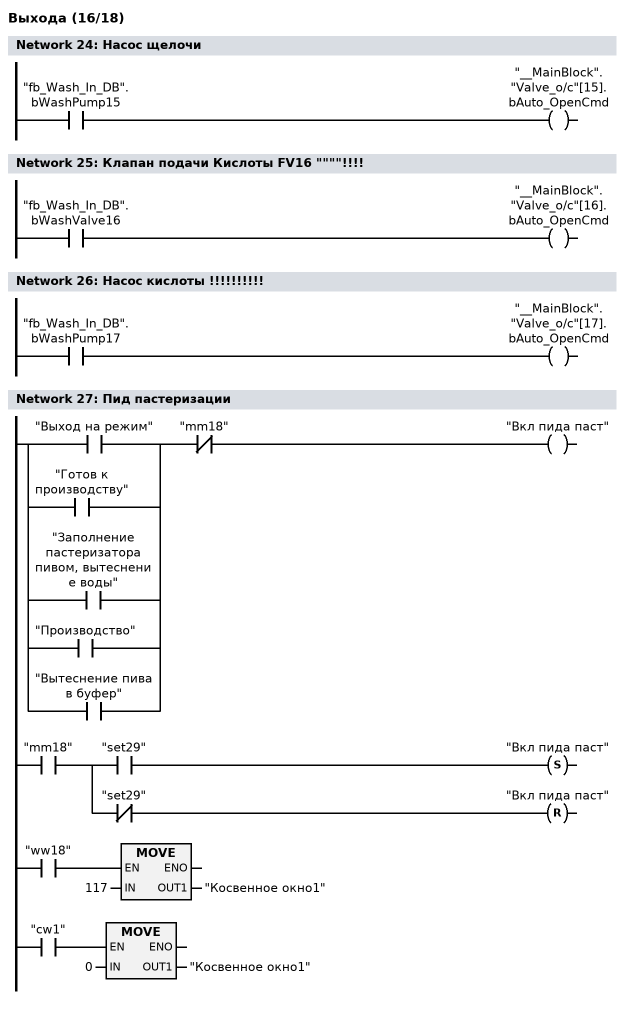
   RUNG wire#powerrail
      Contact( "fb_Wash_In_DB".bWashPump15 )
      Coil( "__MainBlock"."Valve_o/c"[15].bAuto_OpenCmd )
   END_RUNG
   // the same network as SCL:
   "__MainBlock"."Valve_o/c"[15].bAuto_OpenCmd := "fb_Wash_In_DB".bWashPump15;
END_REGION

REGION Network 25: Клапан подачи Кислоты FV16 """"!!!!
   RUNG wire#powerrail
      Contact( "fb_Wash_In_DB".bWashValve16 )
      Coil( "__MainBlock"."Valve_o/c"[16].bAuto_OpenCmd )
   END_RUNG
   // the same network as SCL:
   "__MainBlock"."Valve_o/c"[16].bAuto_OpenCmd := "fb_Wash_In_DB".bWashValve16;
END_REGION

REGION Network 26: Насос кислоты !!!!!!!!!!
   RUNG wire#powerrail
      Contact( "fb_Wash_In_DB".bWashPump17 )
      Coil( "__MainBlock"."Valve_o/c"[17].bAuto_OpenCmd )
   END_RUNG
   // the same network as SCL:
   "__MainBlock"."Valve_o/c"[17].bAuto_OpenCmd := "fb_Wash_In_DB".bWashPump17;
END_REGION

REGION Network 27: Пид пастеризации
   RUNG wire#powerrail
      Contact( "Выход на режим" )
      wire#w1
      I_Contact( "mm18" )
      Coil( "Вкл пида паст" )
   END_RUNG
   RUNG wire#powerrail
      Contact( "Готов к производству" )
   END_RUNG wire#w1
   RUNG wire#powerrail
      Contact( "Заполнение пастеризатора пивом, вытеснение воды" )
   END_RUNG wire#w1
   RUNG wire#powerrail
      Contact( "Производство" )
   END_RUNG wire#w1
   RUNG wire#powerrail
      Contact( "Вытеснение пива в буфер" )
   END_RUNG wire#w1
   RUNG wire#powerrail
      Contact( "mm18" )
      wire#w2
      Contact( "set29" )
      S_Coil( "Вкл пида паст" )
   END_RUNG
   RUNG wire#w2
      I_Contact( "set29" )
      R_Coil( "Вкл пида паст" )
   END_RUNG
   RUNG wire#powerrail
      Contact( "ww18" )
      Move(in := 117, out1 => "Косвенное окно1")
   END_RUNG
   RUNG wire#powerrail
      Contact( "cw1" )
      Move(in := 0, out1 => "Косвенное окно1")
   END_RUNG
   // the same network as SCL:
   "Вкл пида паст" := ("Выход на режим" OR "Готов к производству" OR "Заполнение пастеризатора пивом, вытеснение воды" OR "Производство" OR "Вытеснение пива в буфер") AND NOT "mm18";
   IF "mm18" AND "set29" THEN "Вкл пида паст" := TRUE; END_IF;
   IF "mm18" AND NOT "set29" THEN "Вкл пида паст" := FALSE; END_IF;
   IF "ww18" THEN "Косвенное окно1" := 117; END_IF;
   IF "cw1" THEN "Косвенное окно1" := 0; END_IF;
END_REGION

REGION Network 28: Пид охлаждения
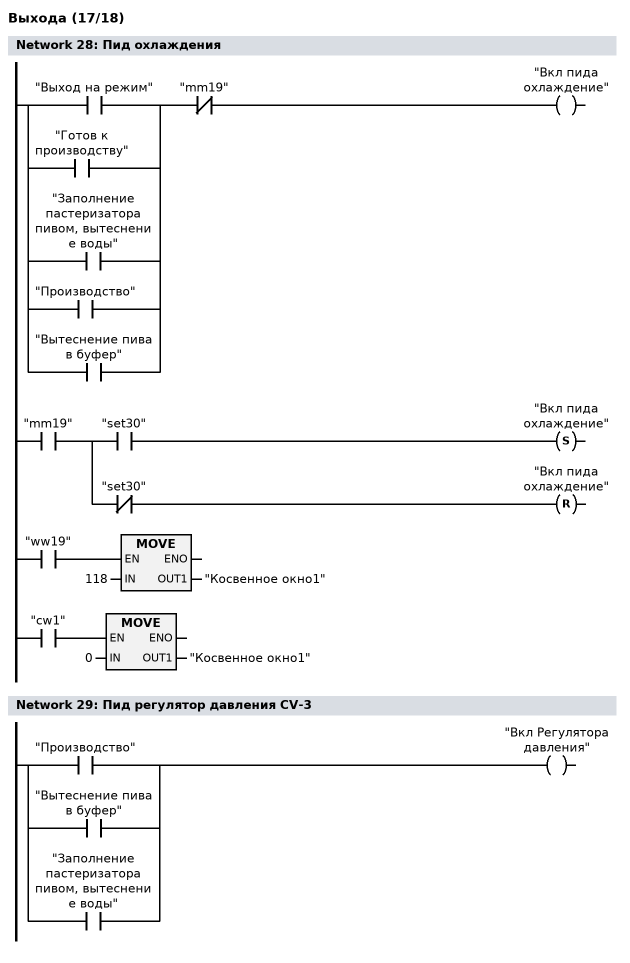
   RUNG wire#powerrail
      Contact( "Выход на режим" )
      wire#w1
      I_Contact( "mm19" )
      Coil( "Вкл пида охлаждение" )
   END_RUNG
   RUNG wire#powerrail
      Contact( "Готов к производству" )
   END_RUNG wire#w1
   RUNG wire#powerrail
      Contact( "Заполнение пастеризатора пивом, вытеснение воды" )
   END_RUNG wire#w1
   RUNG wire#powerrail
      Contact( "Производство" )
   END_RUNG wire#w1
   RUNG wire#powerrail
      Contact( "Вытеснение пива в буфер" )
   END_RUNG wire#w1
   RUNG wire#powerrail
      Contact( "mm19" )
      wire#w2
      Contact( "set30" )
      S_Coil( "Вкл пида охлаждение" )
   END_RUNG
   RUNG wire#w2
      I_Contact( "set30" )
      R_Coil( "Вкл пида охлаждение" )
   END_RUNG
   RUNG wire#powerrail
      Contact( "ww19" )
      Move(in := 118, out1 => "Косвенное окно1")
   END_RUNG
   RUNG wire#powerrail
      Contact( "cw1" )
      Move(in := 0, out1 => "Косвенное окно1")
   END_RUNG
   // the same network as SCL:
   "Вкл пида охлаждение" := ("Выход на режим" OR "Готов к производству" OR "Заполнение пастеризатора пивом, вытеснение воды" OR "Производство" OR "Вытеснение пива в буфер") AND NOT "mm19";
   IF "mm19" AND "set30" THEN "Вкл пида охлаждение" := TRUE; END_IF;
   IF "mm19" AND NOT "set30" THEN "Вкл пида охлаждение" := FALSE; END_IF;
   IF "ww19" THEN "Косвенное окно1" := 118; END_IF;
   IF "cw1" THEN "Косвенное окно1" := 0; END_IF;
END_REGION

REGION Network 29: Пид регулятор давления CV-3
   RUNG wire#powerrail
      Contact( "Производство" )
      wire#w1
      Coil( "Вкл Регулятора давления" )
   END_RUNG
   RUNG wire#powerrail
      Contact( "Вытеснение пива в буфер" )
   END_RUNG wire#w1
   RUNG wire#powerrail
      Contact( "Заполнение пастеризатора пивом, вытеснение воды" )
   END_RUNG wire#w1
   // the same network as SCL:
   "Вкл Регулятора давления" := "Производство" OR "Вытеснение пива в буфер" OR "Заполнение пастеризатора пивом, вытеснение воды";
END_REGION

REGION Network 30: Пид произовдительности М1=М2
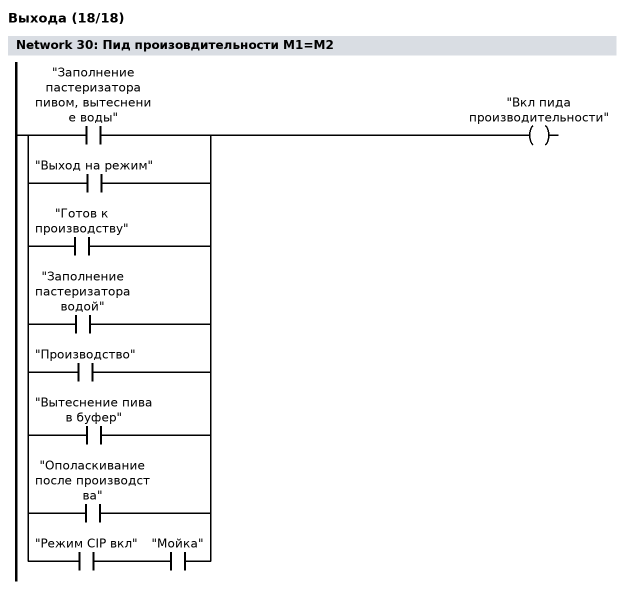
   RUNG wire#powerrail
      Contact( "Заполнение пастеризатора пивом, вытеснение воды" )
      wire#w1
      Coil( "Вкл пида производительности" )
   END_RUNG
   RUNG wire#powerrail
      Contact( "Выход на режим" )
   END_RUNG wire#w1
   RUNG wire#powerrail
      Contact( "Готов к производству" )
   END_RUNG wire#w1
   RUNG wire#powerrail
      Contact( "Заполнение пастеризатора водой" )
   END_RUNG wire#w1
   RUNG wire#powerrail
      Contact( "Производство" )
   END_RUNG wire#w1
   RUNG wire#powerrail
      Contact( "Вытеснение пива в буфер" )
   END_RUNG wire#w1
   RUNG wire#powerrail
      Contact( "Ополаскивание после производства" )
   END_RUNG wire#w1
   RUNG wire#powerrail
      Contact( "Режим СIP вкл" )
      Contact( "Мойка" )
   END_RUNG wire#w1
   // the same network as SCL:
   "Вкл пида производительности" := "Заполнение пастеризатора пивом, вытеснение воды" OR "Выход на режим" OR "Готов к производству" OR "Заполнение пастеризатора водой" OR "Производство" OR "Вытеснение пива в буфер" OR "Ополаскивание после производства" OR ("Режим СIP вкл" AND "Мойка");
END_REGION
END_ORGANIZATION_BLOCK

ORGANIZATION_BLOCK "Реж_Пастеризация пива"   // OB126, LAD, ProgramCycle
TITLE = "Main Program Sweep (Cycle)"
{ S7_Optimized_Access := 'TRUE' }
VERSION : 0.1
   VAR_INPUT
      Initial_Call : Bool;   // Initial call of this OB
      Remanence : Bool;   // =True, if remanent data are available
   END_VAR
BEGIN

REGION Network 1: Заполнение пивом
   // временно привязал переменные на прямую без обработки сигналов DI - ИСПРАВИТЬ!!!!!
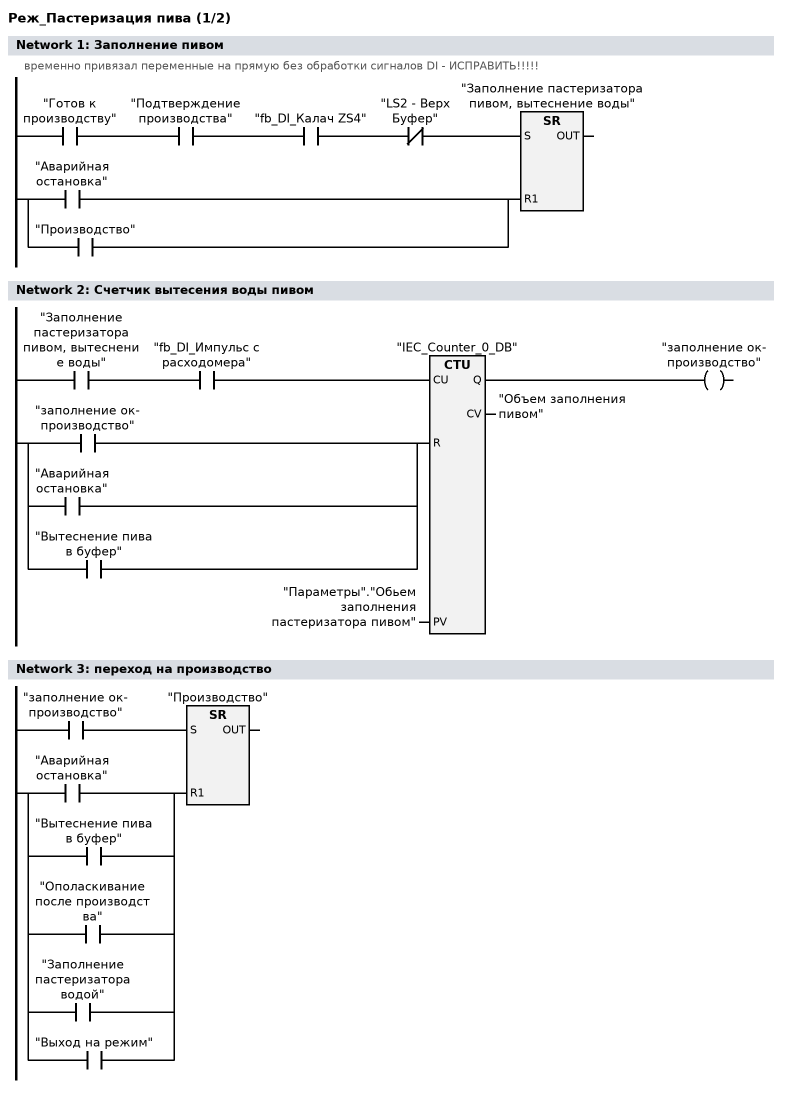
   RUNG wire#powerrail
      Contact( "Готов к производству" )
      Contact( "Подтверждение производства" )
      Contact( "fb_DI_Калач ZS4" )
      I_Contact( "LS2 - Верх Буфер" )
      S_SR(operand := "Заполнение пастеризатора пивом, вытеснение воды", r1 := wire#w1)
   END_RUNG
   RUNG wire#powerrail
      Contact( "Аварийная остановка" )
   END_RUNG wire#w1
   RUNG wire#powerrail
      Contact( "Производство" )
   END_RUNG wire#w1
   // the same network as SCL:
   IF "Готов к производству" AND "Подтверждение производства" AND "fb_DI_Калач ZS4" AND NOT "LS2 - Верх Буфер" THEN
       "Заполнение пастеризатора пивом, вытеснение воды" := TRUE;   // SR flip-flop
   END_IF;
   IF "Аварийная остановка" OR "Производство" THEN
       "Заполнение пастеризатора пивом, вытеснение воды" := FALSE;
   END_IF;
END_REGION

REGION Network 2: Счетчик вытесения воды пивом
   "IEC_Counter_0_DB".CTU(CU := "Заполнение пастеризатора пивом, вытеснение воды" AND "fb_DI_Импульс с расходомера",
                          R := "заполнение ок- производство" OR "Аварийная остановка" OR "Вытеснение пива в буфер",
                          PV := "Параметры"."Обьем заполнения пастеризатора пивом",
                          CV => "Объем заполнения пивом");
   "заполнение ок- производство" := "IEC_Counter_0_DB".Q;
END_REGION

REGION Network 3: переход на производство
   RUNG wire#powerrail
      Contact( "заполнение ок- производство" )
      S_SR(operand := "Производство", r1 := wire#w1)
   END_RUNG
   RUNG wire#powerrail
      Contact( "Аварийная остановка" )
   END_RUNG wire#w1
   RUNG wire#powerrail
      Contact( "Вытеснение пива в буфер" )
   END_RUNG wire#w1
   RUNG wire#powerrail
      Contact( "Ополаскивание после производства" )
   END_RUNG wire#w1
   RUNG wire#powerrail
      Contact( "Заполнение пастеризатора водой" )
   END_RUNG wire#w1
   RUNG wire#powerrail
      Contact( "Выход на режим" )
   END_RUNG wire#w1
   // the same network as SCL:
   IF "заполнение ок- производство" THEN
       "Производство" := TRUE;   // SR flip-flop
   END_IF;
   IF "Аварийная остановка" OR "Вытеснение пива в буфер" OR "Ополаскивание после производства" OR "Заполнение пастеризатора водой" OR "Выход на режим" THEN
       "Производство" := FALSE;
   END_IF;
END_REGION

REGION Network 4: Счетчик объема пастеризации
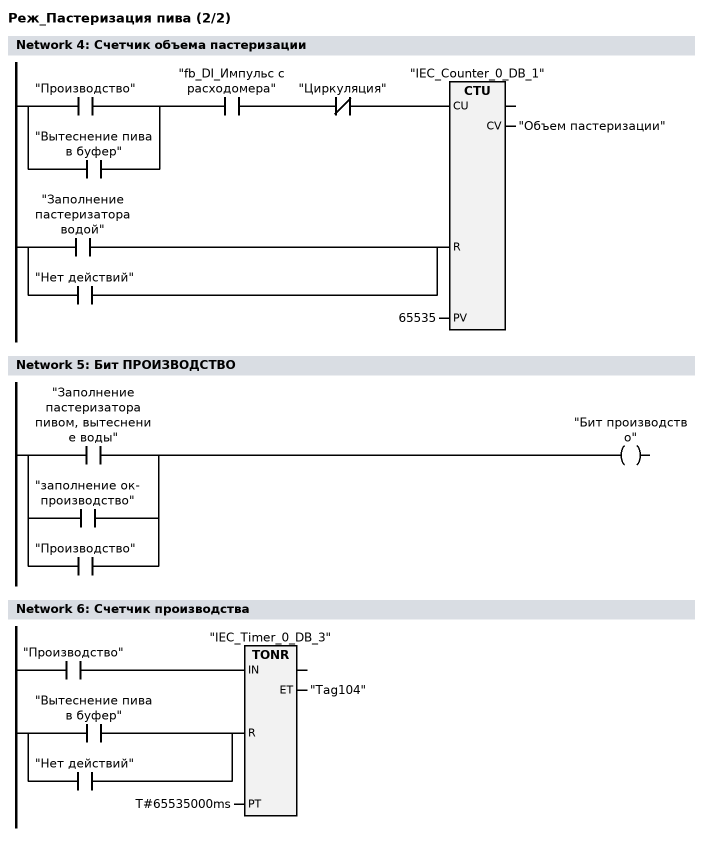
   "IEC_Counter_0_DB_1".CTU(CU := ("Производство" OR "Вытеснение пива в буфер") AND "fb_DI_Импульс с расходомера" AND NOT "Циркуляция",
                           R := "Заполнение пастеризатора водой" OR "Нет действий",
                           PV := 65535,
                           CV => "Объем пастеризации");
END_REGION

REGION Network 5: Бит ПРОИЗВОДСТВО
   RUNG wire#powerrail
      Contact( "Заполнение пастеризатора пивом, вытеснение воды" )
      wire#w1
      Coil( "Бит производство" )
   END_RUNG
   RUNG wire#powerrail
      Contact( "заполнение ок- производство" )
   END_RUNG wire#w1
   RUNG wire#powerrail
      Contact( "Производство" )
   END_RUNG wire#w1
   // the same network as SCL:
   "Бит производство" := "Заполнение пастеризатора пивом, вытеснение воды" OR "заполнение ок- производство" OR "Производство";
END_REGION

REGION Network 6: Счетчик производства
   "IEC_Timer_0_DB_3".TONR(IN := "Производство",
                           R := "Вытеснение пива в буфер" OR "Нет действий",
                           PT := T#65535000ms,
                           ET => "Tag104");
END_REGION
END_ORGANIZATION_BLOCK

ORGANIZATION_BLOCK "Реж_Вытеснение"   // OB127, LAD, ProgramCycle
TITLE = "Main Program Sweep (Cycle)"
{ S7_Optimized_Access := 'TRUE' }
VERSION : 0.1
   VAR_INPUT
      Initial_Call : Bool;   // Initial call of this OB
      Remanence : Bool;   // =True, if remanent data are available
   END_VAR
BEGIN

REGION Network 1: Вытеснение пива в буфер
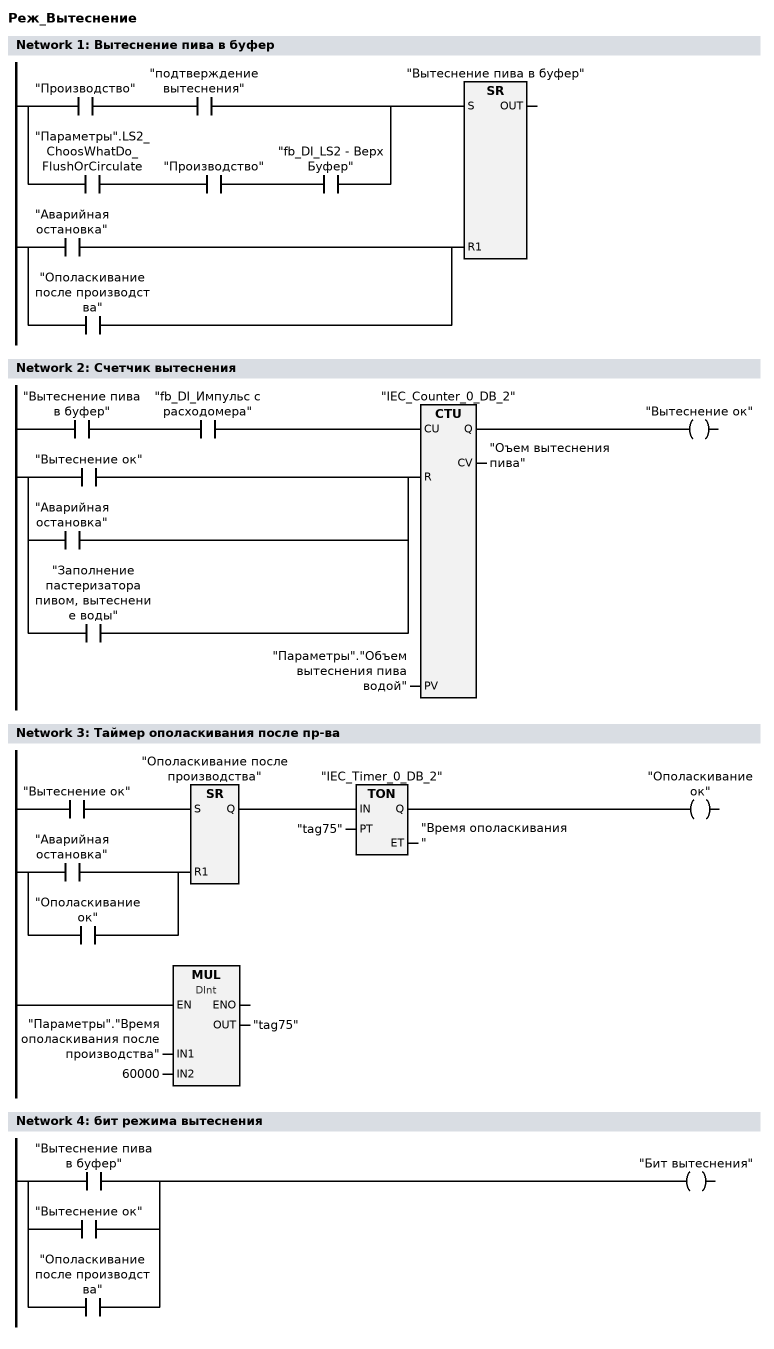
   RUNG wire#powerrail
      Contact( "Производство" )
      Contact( "подтверждение вытеснения" )
      wire#w1
      S_SR(operand := "Вытеснение пива в буфер", r1 := wire#w2)
   END_RUNG
   RUNG wire#powerrail
      Contact( "Параметры".LS2_ChoosWhatDo_FlushOrCirculate )
      Contact( "Производство" )
      Contact( "fb_DI_LS2 - Верх Буфер" )
   END_RUNG wire#w1
   RUNG wire#powerrail
      Contact( "Аварийная остановка" )
   END_RUNG wire#w2
   RUNG wire#powerrail
      Contact( "Ополаскивание после производства" )
   END_RUNG wire#w2
   // the same network as SCL:
   IF ("Производство" AND "подтверждение вытеснения") OR ("Параметры".LS2_ChoosWhatDo_FlushOrCirculate AND "Производство" AND "fb_DI_LS2 - Верх Буфер") THEN
       "Вытеснение пива в буфер" := TRUE;   // SR flip-flop
   END_IF;
   IF "Аварийная остановка" OR "Ополаскивание после производства" THEN
       "Вытеснение пива в буфер" := FALSE;
   END_IF;
END_REGION

REGION Network 2: Счетчик вытеснения
   "IEC_Counter_0_DB_2".CTU(CU := "Вытеснение пива в буфер" AND "fb_DI_Импульс с расходомера",
                           R := "Вытеснение ок" OR "Аварийная остановка" OR "Заполнение пастеризатора пивом, вытеснение воды",
                           PV := "Параметры"."Объем вытеснения пива водой",
                           CV => "Оъем вытеснения пива");
   "Вытеснение ок" := "IEC_Counter_0_DB_2".Q;
END_REGION

REGION Network 3: Таймер ополаскивания после пр-ва
   IF "Вытеснение ок" THEN
       "Ополаскивание после производства" := TRUE;   // SR flip-flop
   END_IF;
   IF "Аварийная остановка" OR "Ополаскивание ок" THEN "Ополаскивание после производства" := FALSE; END_IF;
   "IEC_Timer_0_DB_2".TON(IN := "Ополаскивание после производства", PT := "tag75", ET => "Время ополаскивания");
   "Ополаскивание ок" := "IEC_Timer_0_DB_2".Q;
   "tag75" := "Параметры"."Время ополаскивания после производства" * 60000;
END_REGION

REGION Network 4: бит режима вытеснения
   RUNG wire#powerrail
      Contact( "Вытеснение пива в буфер" )
      wire#w1
      Coil( "Бит вытеснения" )
   END_RUNG
   RUNG wire#powerrail
      Contact( "Вытеснение ок" )
   END_RUNG wire#w1
   RUNG wire#powerrail
      Contact( "Ополаскивание после производства" )
   END_RUNG wire#w1
   // the same network as SCL:
   "Бит вытеснения" := "Вытеснение пива в буфер" OR "Вытеснение ок" OR "Ополаскивание после производства";
END_REGION
END_ORGANIZATION_BLOCK

ORGANIZATION_BLOCK "Реж_Мойка сипом"   // OB128, LAD, ProgramCycle
TITLE = "Main Program Sweep (Cycle)"
{ S7_Optimized_Access := 'TRUE' }
VERSION : 0.1
   VAR_INPUT
      Initial_Call : Bool;   // Initial call of this OB
      Remanence : Bool;   // =True, if remanent data are available
   END_VAR
BEGIN

REGION Network 1: Старт Мойка
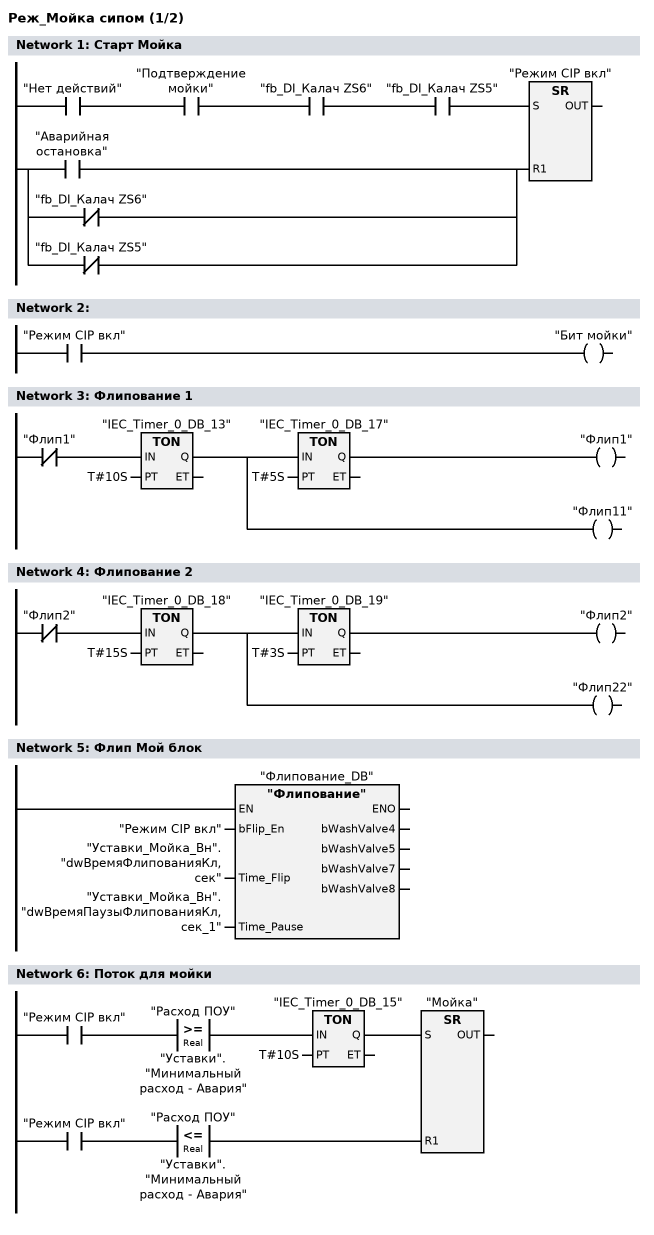
   RUNG wire#powerrail
      Contact( "Нет действий" )
      Contact( "Подтверждение мойки" )
      Contact( "fb_DI_Калач ZS6" )
      Contact( "fb_DI_Калач ZS5" )
      S_SR(operand := "Режим СIP вкл", r1 := wire#w1)
   END_RUNG
   RUNG wire#powerrail
      Contact( "Аварийная остановка" )
   END_RUNG wire#w1
   RUNG wire#powerrail
      I_Contact( "fb_DI_Калач ZS6" )
   END_RUNG wire#w1
   RUNG wire#powerrail
      I_Contact( "fb_DI_Калач ZS5" )
   END_RUNG wire#w1
   // the same network as SCL:
   IF "Нет действий" AND "Подтверждение мойки" AND "fb_DI_Калач ZS6" AND "fb_DI_Калач ZS5" THEN
       "Режим СIP вкл" := TRUE;   // SR flip-flop
   END_IF;
   IF "Аварийная остановка" OR NOT "fb_DI_Калач ZS6" OR NOT "fb_DI_Калач ZS5" THEN
       "Режим СIP вкл" := FALSE;
   END_IF;
END_REGION

REGION Network 2
   RUNG wire#powerrail
      Contact( "Режим СIP вкл" )
      Coil( "Бит мойки" )
   END_RUNG
   // the same network as SCL:
   "Бит мойки" := "Режим СIP вкл";
END_REGION

REGION Network 3: Флипование 1
   "IEC_Timer_0_DB_13".TON(IN := NOT "Флип1", PT := T#10S);
   "IEC_Timer_0_DB_17".TON(IN := "IEC_Timer_0_DB_13".Q, PT := T#5S);
   "Флип1" := "IEC_Timer_0_DB_17".Q;
   "Флип11" := "IEC_Timer_0_DB_13".Q;
END_REGION

REGION Network 4: Флипование 2
   "IEC_Timer_0_DB_18".TON(IN := NOT "Флип2", PT := T#15S);
   "IEC_Timer_0_DB_19".TON(IN := "IEC_Timer_0_DB_18".Q, PT := T#3S);
   "Флип2" := "IEC_Timer_0_DB_19".Q;
   "Флип22" := "IEC_Timer_0_DB_18".Q;
END_REGION

REGION Network 5: Флип Мой блок
   RUNG wire#powerrail
      "Флипование_DB"(bFlip_En := "Режим СIP вкл", Time_Flip := "Уставки_Мойка_Вн"."dwВремяФлипованияКл,сек", Time_Pause := "Уставки_Мойка_Вн"."dwВремяПаузыФлипованияКл,сек_1", bWashValve4 =>, bWashValve5 =>, bWashValve7 =>, bWashValve8 =>)
   END_RUNG
   // the same network as SCL:
   "Флипование_DB"(bFlip_En := "Режим СIP вкл",   // "Флипование"
                   Time_Flip := "Уставки_Мойка_Вн"."dwВремяФлипованияКл,сек",
                   Time_Pause := "Уставки_Мойка_Вн"."dwВремяПаузыФлипованияКл,сек_1");
END_REGION

REGION Network 6: Поток для мойки
   "IEC_Timer_0_DB_15".TON(IN := "Режим СIP вкл" AND ("Расход ПОУ" >= "Уставки"."Минимальный расход - Авария"),
                           PT := T#10S);
   IF "IEC_Timer_0_DB_15".Q THEN
       "Мойка" := TRUE;   // SR flip-flop
   END_IF;
   IF "Режим СIP вкл" AND ("Расход ПОУ" <= "Уставки"."Минимальный расход - Авария") THEN
       "Мойка" := FALSE;
   END_IF;
END_REGION

REGION Network 7: НЕт расхода при мойке СИП
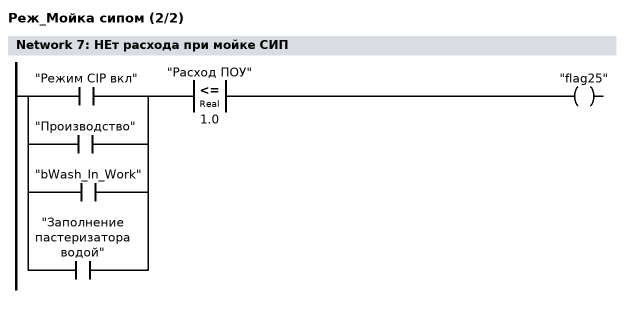
   RUNG wire#powerrail
      Contact( "Режим СIP вкл" )
      wire#w1
      { S7_Templates := "SrcType := Real" } LE_Contact(in1 := "Расход ПОУ", in2 := 1.0)
      Coil( "flag25" )
   END_RUNG
   RUNG wire#powerrail
      Contact( "Производство" )
   END_RUNG wire#w1
   RUNG wire#powerrail
      Contact( "bWash_In_Work" )
   END_RUNG wire#w1
   RUNG wire#powerrail
      Contact( "Заполнение пастеризатора водой" )
   END_RUNG wire#w1
   // the same network as SCL:
   "flag25" := ("Режим СIP вкл" OR "Производство" OR "bWash_In_Work" OR "Заполнение пастеризатора водой") AND ("Расход ПОУ" <= 1.0);
END_REGION
END_ORGANIZATION_BLOCK

ORGANIZATION_BLOCK "ПИД"   // OB129, LAD, ProgramCycle
TITLE = "Main Program Sweep (Cycle)"
{ S7_Optimized_Access := 'TRUE' }
VERSION : 0.1
   VAR_INPUT
      Initial_Call : Bool;   // Initial call of this OB
      Remanence : Bool;   // =True, if remanent data are available
   END_VAR
BEGIN

REGION Network 1: ПИД - Нагрев
   // ПИД нагрева уставка при мойке и при Пастеризации
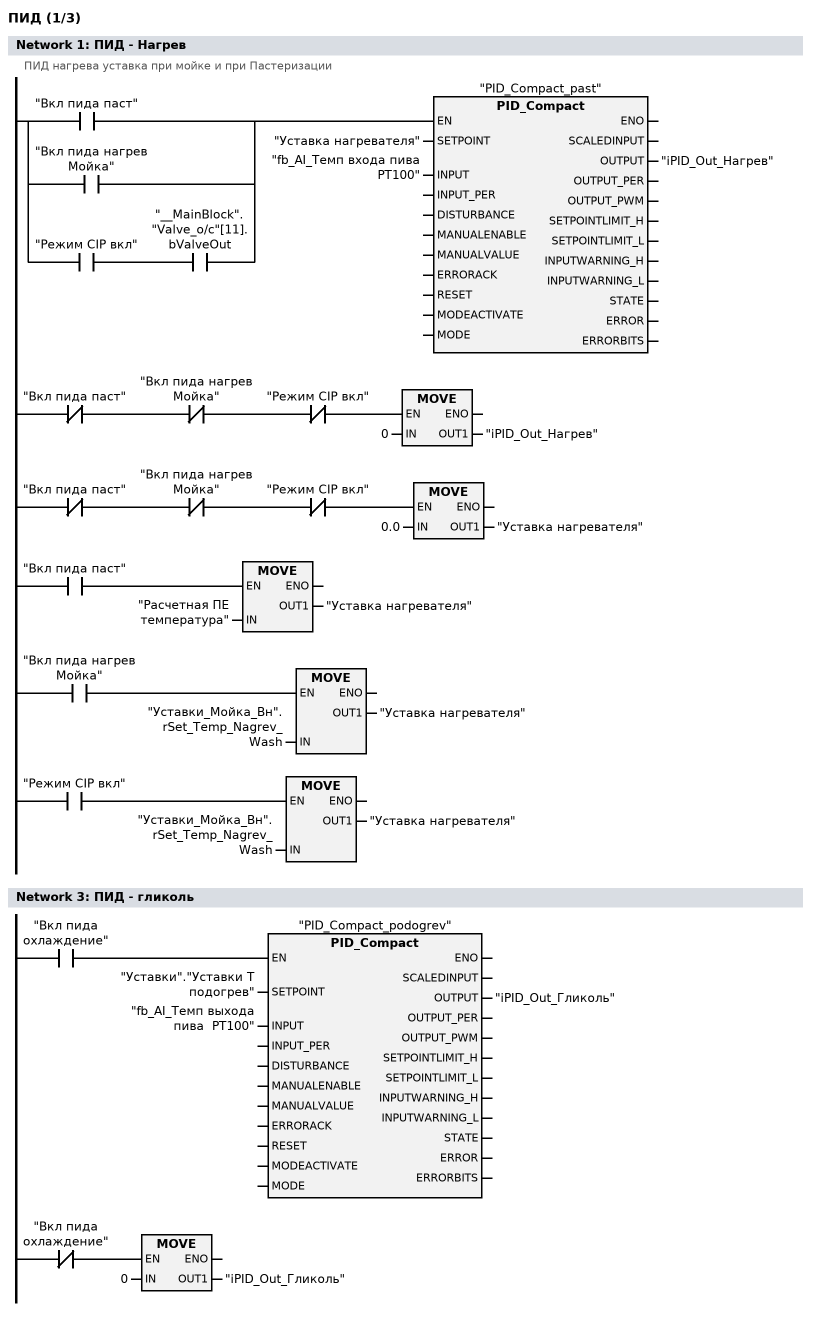
   IF "Вкл пида паст" OR "Вкл пида нагрев Мойка" OR ("Режим СIP вкл" AND "__MainBlock"."Valve_o/c"[11].bValveOut) THEN
       "PID_Compact_past"(Setpoint := "Уставка нагревателя",   // PID_Compact
                          Input := "fb_AI_Темп входа пива PT100",
                          Output => "iPID_Out_Нагрев");
   END_IF;
   IF NOT "Вкл пида паст" AND NOT "Вкл пида нагрев Мойка" AND NOT "Режим СIP вкл" THEN
       "iPID_Out_Нагрев" := 0;
       "Уставка нагревателя" := 0.0;
   END_IF;
   IF "Вкл пида паст" THEN "Уставка нагревателя" := "Расчетная ПЕ температура"; END_IF;
   IF "Вкл пида нагрев Мойка" THEN "Уставка нагревателя" := "Уставки_Мойка_Вн".rSet_Temp_Nagrev_Wash; END_IF;
   IF "Режим СIP вкл" THEN "Уставка нагревателя" := "Уставки_Мойка_Вн".rSet_Temp_Nagrev_Wash; END_IF;
END_REGION

REGION Network 2 (SCL): Коэффициэнты ПИД-1
   // Нагрев
   // Коэфициент_s

   "PID_Compact_past".Retain.CtrlParams.Gain := "__MainBlock".PID[1].k_p;
   "PID_Compact_past".Retain.CtrlParams.Ti := "__MainBlock".PID[1].k_I;
   "PID_Compact_past".Retain.CtrlParams.Td := "__MainBlock".PID[1].k_D;
END_REGION

REGION Network 3: ПИД - гликоль
   IF "Вкл пида охлаждение" THEN
       "PID_Compact_podogrev"(Setpoint := "Уставки"."Уставки Т подогрев",   // PID_Compact
                              Input := "fb_AI_Темп выхода пива  PT100",
                              Output => "iPID_Out_Гликоль");
   END_IF;
   IF NOT "Вкл пида охлаждение" THEN "iPID_Out_Гликоль" := 0; END_IF;
END_REGION

REGION Network 4 (SCL): Коэффициэнты ПИД-2
   // Cooling
   // Коэфициент_s

   "PID_Compact_podogrev".Retain.CtrlParams.Gain := "__MainBlock".PID[2].k_p;
   "PID_Compact_podogrev".Retain.CtrlParams.Ti := "__MainBlock".PID[2].k_I;
   "PID_Compact_podogrev".Retain.CtrlParams.Td := "__MainBlock".PID[2].k_D;
END_REGION

REGION Network 5: Давлени регулятор
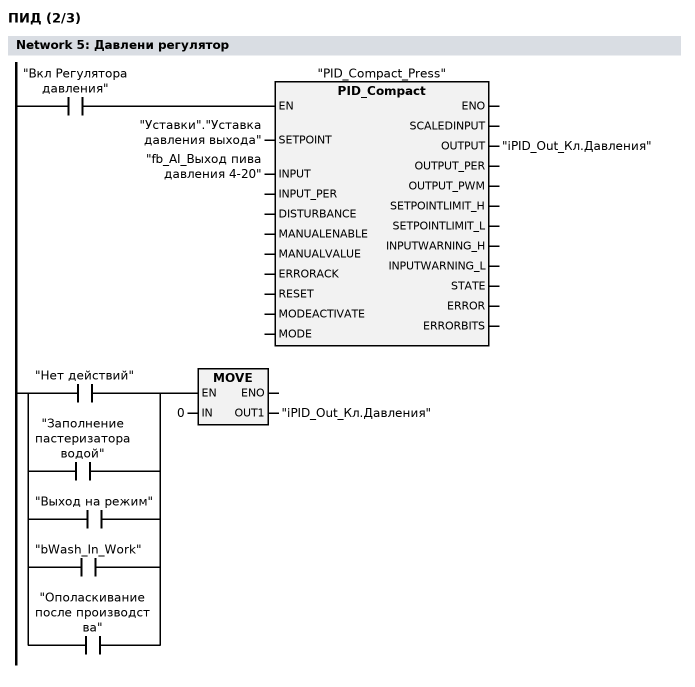
   IF "Вкл Регулятора давления" THEN
       "PID_Compact_Press"(Setpoint := "Уставки"."Уставка давления выхода",   // PID_Compact
                           Input := "fb_AI_Выход пива давления 4-20",
                           Output => "iPID_Out_Кл.Давления");
   END_IF;
   IF "Нет действий" OR "Заполнение пастеризатора водой" OR "Выход на режим" OR "bWash_In_Work" OR "Ополаскивание после производства" THEN
       "iPID_Out_Кл.Давления" := 0;
   END_IF;
END_REGION

REGION Network 6 (SCL): Коэффициэнты ПИД-3
   // Press
   // Коэфициент_s

   "PID_Compact_Press".Retain.CtrlParams.Gain := "__MainBlock".PID[3].k_p;
   "PID_Compact_Press".Retain.CtrlParams.Ti := "__MainBlock".PID[3].k_I;
   "PID_Compact_Press".Retain.CtrlParams.Td := "__MainBlock".PID[3].k_D;
END_REGION

REGION Network 7: ПИД - расход М1/М2
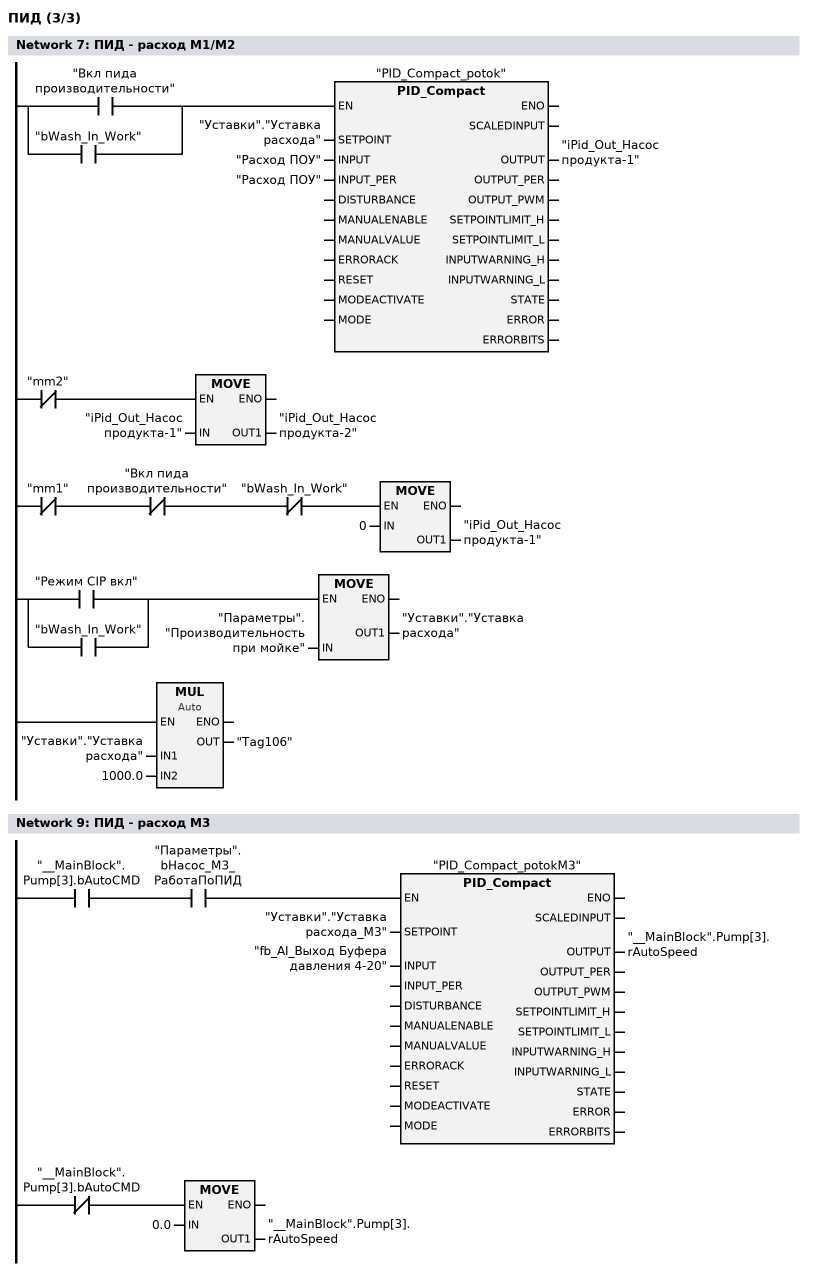
   IF "Вкл пида производительности" OR "bWash_In_Work" THEN
       "PID_Compact_potok"(Setpoint := "Уставки"."Уставка расхода",   // PID_Compact
                           Input := "Расход ПОУ",
                           Input_PER := "Расход ПОУ",
                           Output => "iPid_Out_Насос продукта-1");
   END_IF;
   IF NOT "mm2" THEN "iPid_Out_Насос продукта-2" := "iPid_Out_Насос продукта-1"; END_IF;
   IF NOT "mm1" AND NOT "Вкл пида производительности" AND NOT "bWash_In_Work" THEN
       "iPid_Out_Насос продукта-1" := 0;
   END_IF;
   IF "Режим СIP вкл" OR "bWash_In_Work" THEN
       "Уставки"."Уставка расхода" := "Параметры"."Производительность при мойке";
   END_IF;
   "Tag106" := "Уставки"."Уставка расхода" * 1000.0;
END_REGION

REGION Network 8 (SCL): Коэффициэнты ПИД-4
   // Flow
   // Коэфициент_s

   "PID_Compact_potok".Retain.CtrlParams.Gain := "__MainBlock".PID[4].k_p;
   "PID_Compact_potok".Retain.CtrlParams.Ti := "__MainBlock".PID[4].k_I;
   "PID_Compact_potok".Retain.CtrlParams.Td := "__MainBlock".PID[4].k_D;
END_REGION

REGION Network 9: ПИД - расход М3
   IF "__MainBlock".Pump[3].bAutoCMD AND "Параметры".bНасос_М3_РаботаПоПИД THEN
       "PID_Compact_potokМ3"(Setpoint := "Уставки"."Уставка расхода_М3",   // PID_Compact
                             Input := "fb_AI_Выход Буфера давления 4-20",
                             Output => "__MainBlock".Pump[3].rAutoSpeed);
   END_IF;
   IF NOT "__MainBlock".Pump[3].bAutoCMD THEN "__MainBlock".Pump[3].rAutoSpeed := 0.0; END_IF;
END_REGION

REGION Network 10 (SCL): Коэффициэнты ПИД-5
   // Flow
   // Коэфициент_s

   "PID_Compact_potokМ3".Retain.CtrlParams.Gain := "__MainBlock".PID[5].k_p;
   "PID_Compact_potokМ3".Retain.CtrlParams.Ti := "__MainBlock".PID[5].k_I;
   "PID_Compact_potokМ3".Retain.CtrlParams.Td := "__MainBlock".PID[5].k_D;
END_REGION
END_ORGANIZATION_BLOCK

ORGANIZATION_BLOCK "Время цикла Автомат состояний"   // OB130, LAD, ProgramCycle
TITLE = "Main Program Sweep (Cycle)"
{ S7_Optimized_Access := 'TRUE' }
VERSION : 0.1
   VAR_INPUT
      Initial_Call : Bool;   // Initial call of this OB
      Remanence : Bool;   // =True, if remanent data are available
   END_VAR
BEGIN

REGION Network 1: Пройцесс в мин/сек вывод на экран
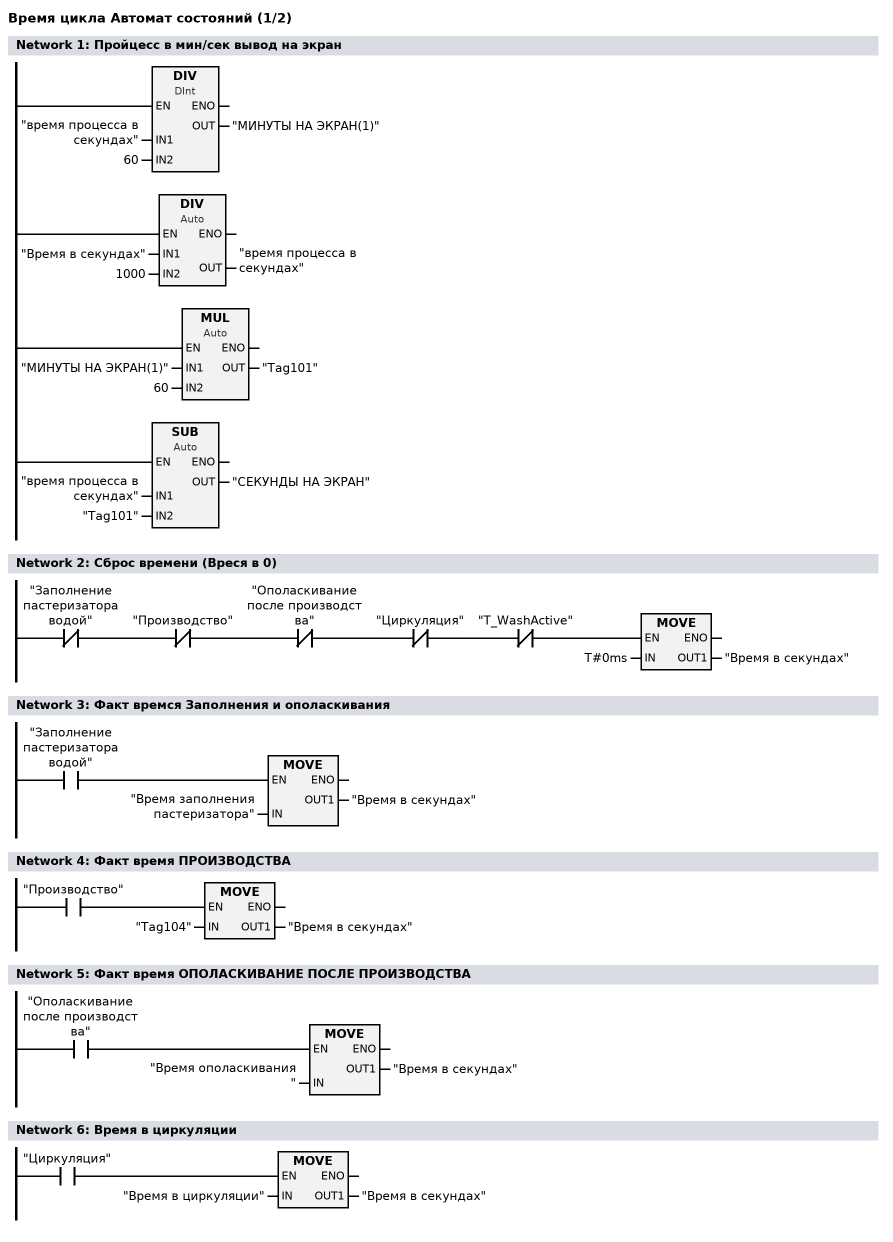
   RUNG wire#powerrail
      { S7_Templates := "SrcType := DInt" } Div(in1 := "время процесса в секундах", in2 := 60, out => "МИНУТЫ НА ЭКРАН(1)")
   END_RUNG
   RUNG wire#powerrail
      Div(in1 := "Время в секундах", in2 := 1000, out => "время процесса в секундах")
   END_RUNG
   RUNG wire#powerrail
      Mul(in1 := "МИНУТЫ НА ЭКРАН(1)", in2 := 60, out => "Tag101")
   END_RUNG
   RUNG wire#powerrail
      Sub(in1 := "время процесса в секундах", in2 := "Tag101", out => "СЕКУНДЫ НА ЭКРАН")
   END_RUNG
   // the same network as SCL:
   "МИНУТЫ НА ЭКРАН(1)" := "время процесса в секундах" / 60;
   "время процесса в секундах" := "Время в секундах" / 1000;
   "Tag101" := "МИНУТЫ НА ЭКРАН(1)" * 60;
   "СЕКУНДЫ НА ЭКРАН" := "время процесса в секундах" - "Tag101";
END_REGION

REGION Network 2: Сброс времени (Вреся в 0)
   RUNG wire#powerrail
      I_Contact( "Заполнение пастеризатора водой" )
      I_Contact( "Производство" )
      I_Contact( "Ополаскивание после производства" )
      I_Contact( "Циркуляция" )
      I_Contact( "T_WashActive" )
      Move(in := T#0ms, out1 => "Время в секундах")
   END_RUNG
   // the same network as SCL:
   IF NOT "Заполнение пастеризатора водой" AND NOT "Производство" AND NOT "Ополаскивание после производства" AND NOT "Циркуляция" AND NOT "T_WashActive" THEN
       "Время в секундах" := T#0ms;
   END_IF;
END_REGION

REGION Network 3: Факт времся Заполнения и ополаскивания
   RUNG wire#powerrail
      Contact( "Заполнение пастеризатора водой" )
      Move(in := "Время заполнения пастеризатора", out1 => "Время в секундах")
   END_RUNG
   // the same network as SCL:
   IF "Заполнение пастеризатора водой" THEN "Время в секундах" := "Время заполнения пастеризатора"; END_IF;
END_REGION

REGION Network 4: Факт время ПРОИЗВОДСТВА
   RUNG wire#powerrail
      Contact( "Производство" )
      Move(in := "Tag104", out1 => "Время в секундах")
   END_RUNG
   // the same network as SCL:
   IF "Производство" THEN "Время в секундах" := "Tag104"; END_IF;
END_REGION

REGION Network 5: Факт время ОПОЛАСКИВАНИЕ ПОСЛЕ ПРОИЗВОДСТВА
   RUNG wire#powerrail
      Contact( "Ополаскивание после производства" )
      Move(in := "Время ополаскивания", out1 => "Время в секундах")
   END_RUNG
   // the same network as SCL:
   IF "Ополаскивание после производства" THEN "Время в секундах" := "Время ополаскивания"; END_IF;
END_REGION

REGION Network 6: Время в циркуляции
   RUNG wire#powerrail
      Contact( "Циркуляция" )
      Move(in := "Время в циркуляции", out1 => "Время в секундах")
   END_RUNG
   // the same network as SCL:
   IF "Циркуляция" THEN "Время в секундах" := "Время в циркуляции"; END_IF;
END_REGION

REGION Network 7: Автомат состояния, номер режима
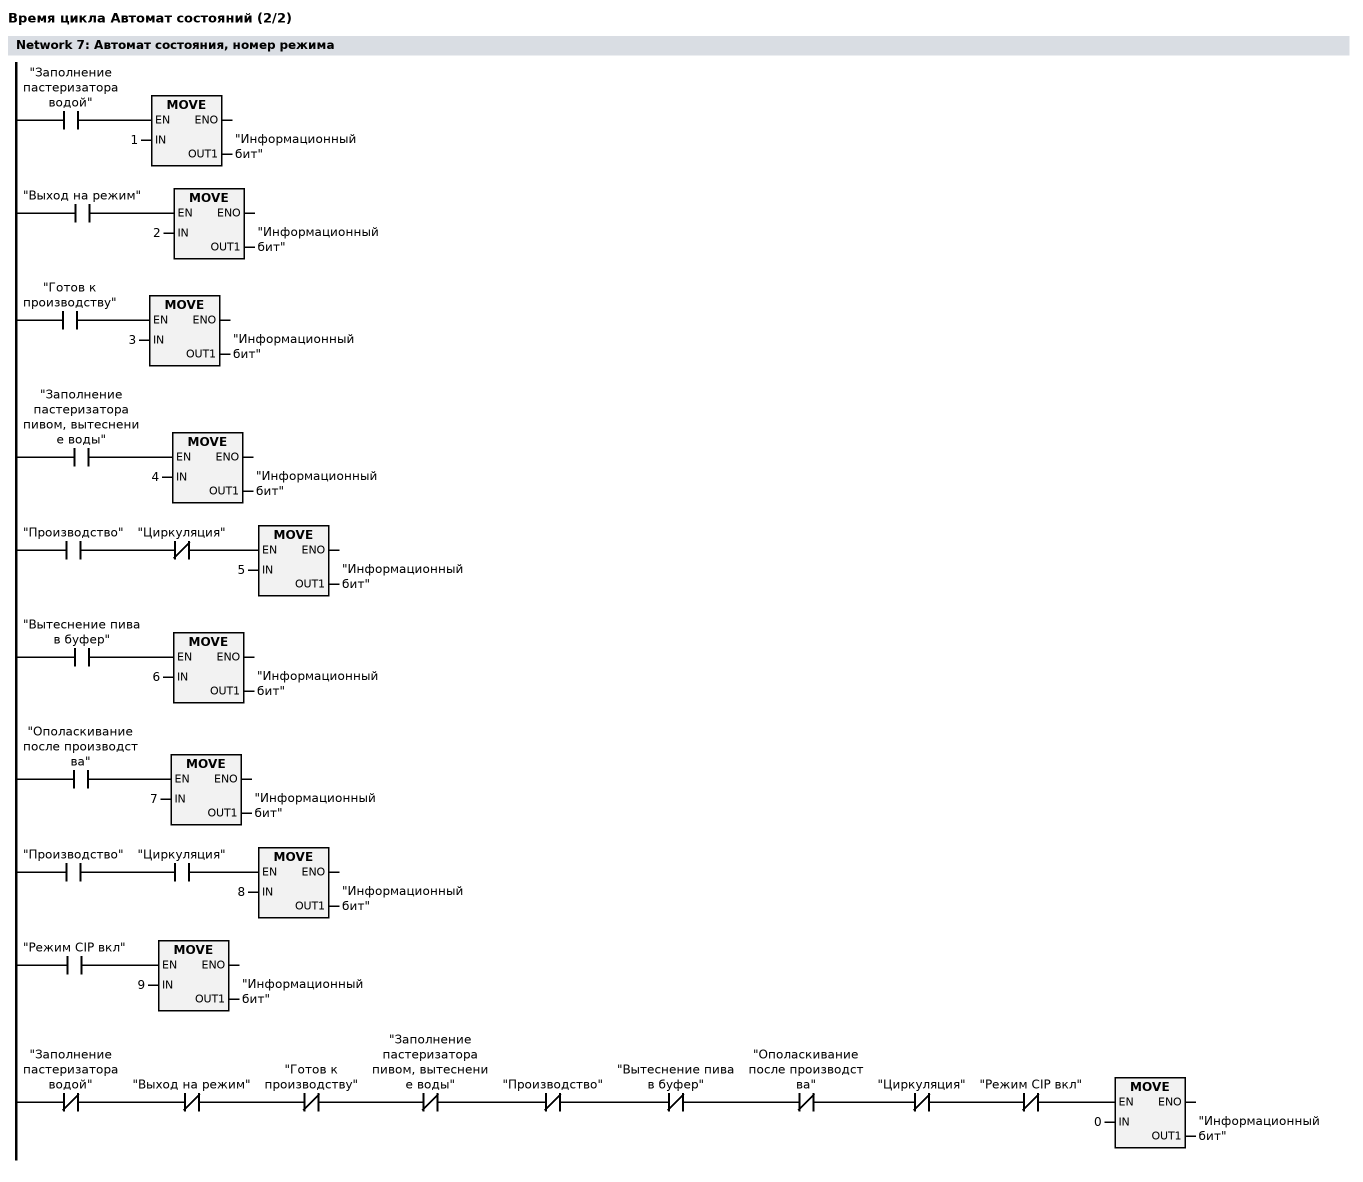
   RUNG wire#powerrail
      Contact( "Заполнение пастеризатора водой" )
      Move(in := 1, out1 => "Информационный бит")
   END_RUNG
   RUNG wire#powerrail
      Contact( "Выход на режим" )
      Move(in := 2, out1 => "Информационный бит")
   END_RUNG
   RUNG wire#powerrail
      Contact( "Готов к производству" )
      Move(in := 3, out1 => "Информационный бит")
   END_RUNG
   RUNG wire#powerrail
      Contact( "Заполнение пастеризатора пивом, вытеснение воды" )
      Move(in := 4, out1 => "Информационный бит")
   END_RUNG
   RUNG wire#powerrail
      Contact( "Производство" )
      I_Contact( "Циркуляция" )
      Move(in := 5, out1 => "Информационный бит")
   END_RUNG
   RUNG wire#powerrail
      Contact( "Вытеснение пива в буфер" )
      Move(in := 6, out1 => "Информационный бит")
   END_RUNG
   RUNG wire#powerrail
      Contact( "Ополаскивание после производства" )
      Move(in := 7, out1 => "Информационный бит")
   END_RUNG
   RUNG wire#powerrail
      Contact( "Производство" )
      Contact( "Циркуляция" )
      Move(in := 8, out1 => "Информационный бит")
   END_RUNG
   RUNG wire#powerrail
      Contact( "Режим СIP вкл" )
      Move(in := 9, out1 => "Информационный бит")
   END_RUNG
   RUNG wire#powerrail
      I_Contact( "Заполнение пастеризатора водой" )
      I_Contact( "Выход на режим" )
      I_Contact( "Готов к производству" )
      I_Contact( "Заполнение пастеризатора пивом, вытеснение воды" )
      I_Contact( "Производство" )
      I_Contact( "Вытеснение пива в буфер" )
      I_Contact( "Ополаскивание после производства" )
      I_Contact( "Циркуляция" )
      I_Contact( "Режим СIP вкл" )
      Move(in := 0, out1 => "Информационный бит")
   END_RUNG
   // the same network as SCL:
   IF "Заполнение пастеризатора водой" THEN "Информационный бит" := 1; END_IF;
   IF "Выход на режим" THEN "Информационный бит" := 2; END_IF;
   IF "Готов к производству" THEN "Информационный бит" := 3; END_IF;
   IF "Заполнение пастеризатора пивом, вытеснение воды" THEN "Информационный бит" := 4; END_IF;
   IF "Производство" AND NOT "Циркуляция" THEN "Информационный бит" := 5; END_IF;
   IF "Вытеснение пива в буфер" THEN "Информационный бит" := 6; END_IF;
   IF "Ополаскивание после производства" THEN "Информационный бит" := 7; END_IF;
   IF "Производство" AND "Циркуляция" THEN "Информационный бит" := 8; END_IF;
   IF "Режим СIP вкл" THEN "Информационный бит" := 9; END_IF;
   IF NOT "Заполнение пастеризатора водой" AND NOT "Выход на режим" AND NOT "Готов к производству" AND NOT "Заполнение пастеризатора пивом, вытеснение воды" AND NOT "Производство" AND NOT "Вытеснение пива в буфер" AND NOT "Ополаскивание после производства" AND NOT "Циркуляция" AND NOT "Режим СIP вкл" THEN
       "Информационный бит" := 0;
   END_IF;
END_REGION
END_ORGANIZATION_BLOCK

ORGANIZATION_BLOCK "Аварии"   // OB131, LAD, ProgramCycle
TITLE = "Main Program Sweep (Cycle)"
{ S7_Optimized_Access := 'TRUE' }
VERSION : 0.1
   VAR_INPUT
      Initial_Call : Bool;   // Initial call of this OB
      Remanence : Bool;   // =True, if remanent data are available
   END_VAR
   VAR_TEMP   // added for the SCL form of the ladder/FBD networks
      _w1 : Bool;
      _w2 : Bool;
      _w3 : Bool;
      _w4 : Bool;
      _w5 : Bool;
   END_VAR
BEGIN

REGION Network 1: Обраотка аварий
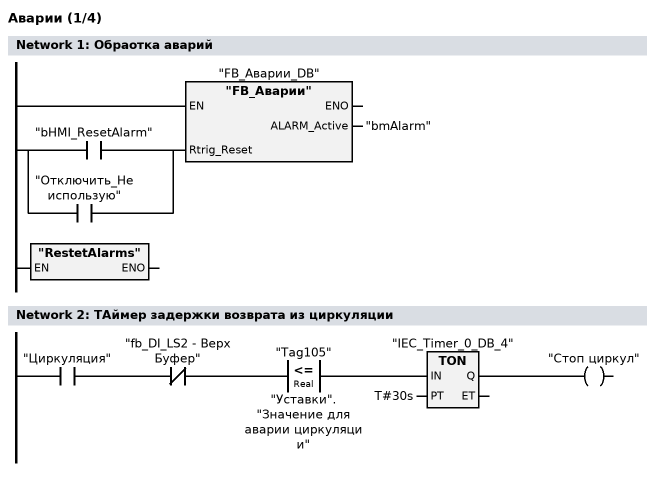
   RUNG wire#powerrail
      "FB_Аварии_DB"(Rtrig_Reset := wire#w1, ALARM_Active => "bmAlarm")
   END_RUNG
   RUNG wire#powerrail
      Contact( "bHMI_ResetAlarm" )
   END_RUNG wire#w1
   RUNG wire#powerrail
      Contact( "Отключить_Не использую" )
   END_RUNG wire#w1
   RUNG wire#powerrail
      "RestetAlarms"()
   END_RUNG
   // the same network as SCL:
   "FB_Аварии_DB"(Rtrig_Reset := "bHMI_ResetAlarm" OR "Отключить_Не использую", ALARM_Active => "bmAlarm");   // "FB_Аварии"
   "RestetAlarms"();
END_REGION

REGION Network 2: ТАймер задержки возврата из циркуляции
   "IEC_Timer_0_DB_4".TON(IN := "Циркуляция" AND NOT "fb_DI_LS2 - Верх Буфер" AND ("Tag105" <= "Уставки"."Значение для аварии циркуляции"),
                          PT := T#30s);
   "Стоп циркул" := "IEC_Timer_0_DB_4".Q;
END_REGION

REGION Network 3: Переход в циркуляцию
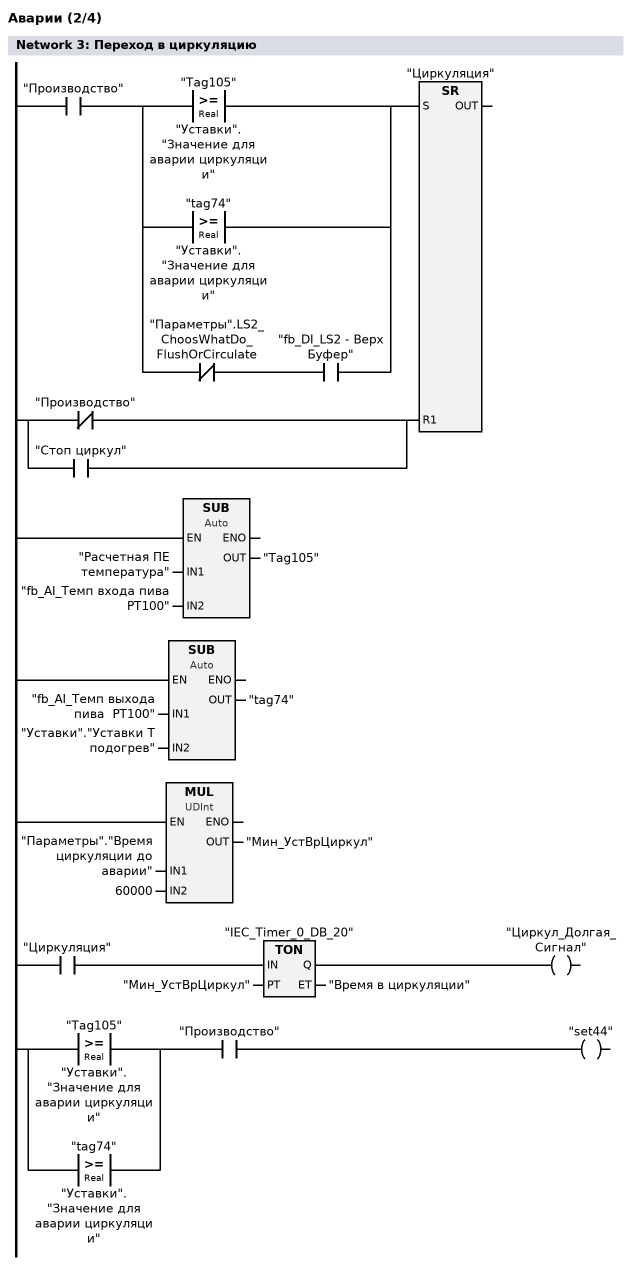
   IF "Производство" AND (("Tag105" >= "Уставки"."Значение для аварии циркуляции") OR ("tag74" >= "Уставки"."Значение для аварии циркуляции") OR (NOT "Параметры".LS2_ChoosWhatDo_FlushOrCirculate AND "fb_DI_LS2 - Верх Буфер")) THEN
       "Циркуляция" := TRUE;   // SR flip-flop
   END_IF;
   IF NOT "Производство" OR "Стоп циркул" THEN "Циркуляция" := FALSE; END_IF;
   "Tag105" := "Расчетная ПЕ температура" - "fb_AI_Темп входа пива PT100";
   "tag74" := "fb_AI_Темп выхода пива  PT100" - "Уставки"."Уставки Т подогрев";
   "Мин_УстВрЦиркул" := "Параметры"."Время циркуляции до аварии" * 60000;
   "IEC_Timer_0_DB_20".TON(IN := "Циркуляция", PT := "Мин_УстВрЦиркул", ET => "Время в циркуляции");
   "Циркул_Долгая_Сигнал" := "IEC_Timer_0_DB_20".Q;
   "set44" := (("Tag105" >= "Уставки"."Значение для аварии циркуляции") OR ("tag74" >= "Уставки"."Значение для аварии циркуляции")) AND "Производство";
END_REGION

REGION Network 4: авария давления секции пастеризации
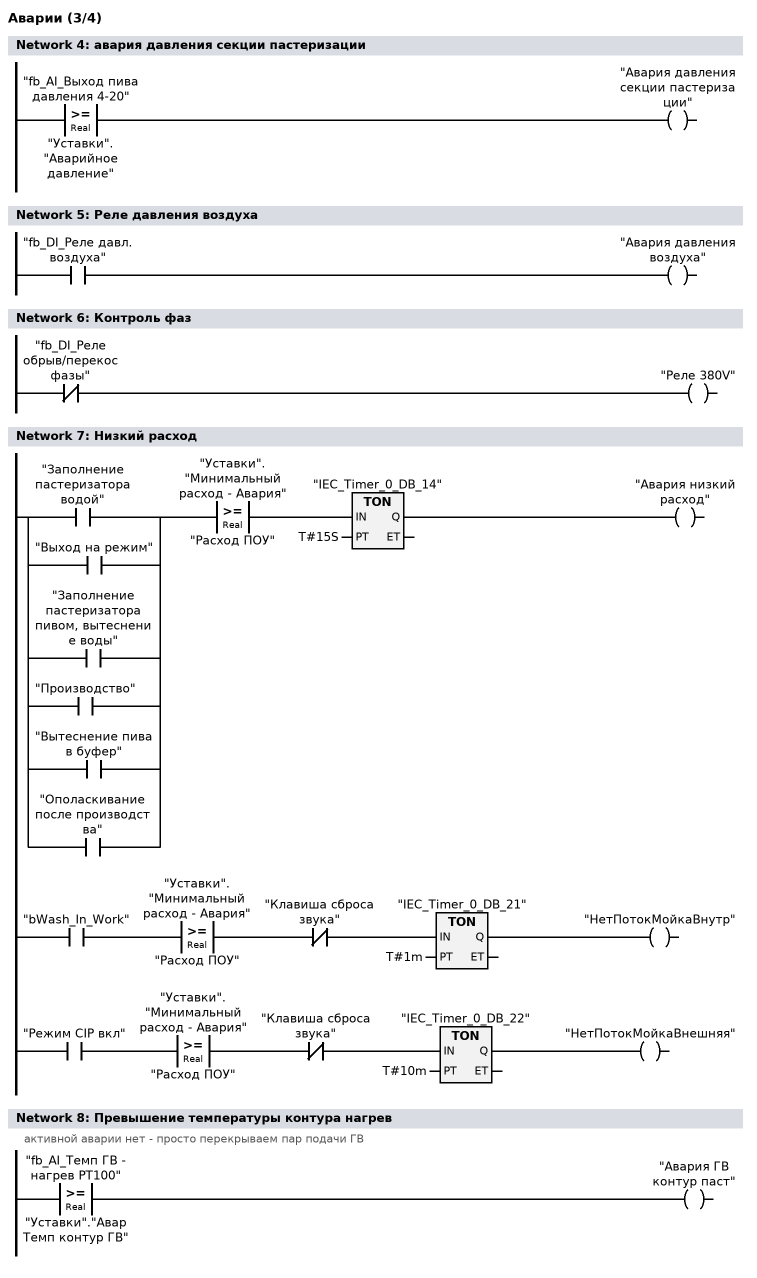
   RUNG wire#powerrail
      { S7_Templates := "SrcType := Real" } GE_Contact(in1 := "fb_AI_Выход пива давления 4-20", in2 := "Уставки"."Аварийное давление")
      Coil( "Авария давления секции пастеризации" )
   END_RUNG
   // the same network as SCL:
   "Авария давления секции пастеризации" := "fb_AI_Выход пива давления 4-20" >= "Уставки"."Аварийное давление";
END_REGION

REGION Network 5: Реле давления воздуха
   RUNG wire#powerrail
      Contact( "fb_DI_Реле давл. воздуха" )
      Coil( "Авария давления воздуха" )
   END_RUNG
   // the same network as SCL:
   "Авария давления воздуха" := "fb_DI_Реле давл. воздуха";
END_REGION

REGION Network 6: Контроль фаз
   RUNG wire#powerrail
      I_Contact( "fb_DI_Реле обрыв/перекос фазы" )
      Coil( "Реле 380V" )
   END_RUNG
   // the same network as SCL:
   "Реле 380V" := NOT "fb_DI_Реле обрыв/перекос фазы";
END_REGION

REGION Network 7: Низкий расход
   "IEC_Timer_0_DB_14".TON(IN := ("Заполнение пастеризатора водой" OR "Выход на режим" OR "Заполнение пастеризатора пивом, вытеснение воды" OR "Производство" OR "Вытеснение пива в буфер" OR "Ополаскивание после производства") AND ("Уставки"."Минимальный расход - Авария" >= "Расход ПОУ"),
                           PT := T#15S);
   "Авария низкий расход" := "IEC_Timer_0_DB_14".Q;
   "IEC_Timer_0_DB_21".TON(IN := "bWash_In_Work" AND ("Уставки"."Минимальный расход - Авария" >= "Расход ПОУ") AND NOT "Клавиша сброса звука",
                           PT := T#1m);
   "НетПотокМойкаВнутр" := "IEC_Timer_0_DB_21".Q;
   "IEC_Timer_0_DB_22".TON(IN := "Режим СIP вкл" AND ("Уставки"."Минимальный расход - Авария" >= "Расход ПОУ") AND NOT "Клавиша сброса звука",
                           PT := T#10m);
   "НетПотокМойкаВнешняя" := "IEC_Timer_0_DB_22".Q;
END_REGION

REGION Network 8: Превышение температуры контура нагрев
   // активной аварии нет - просто перекрываем пар подачи ГВ
   RUNG wire#powerrail
      { S7_Templates := "SrcType := Real" } GE_Contact(in1 := "fb_AI_Темп ГВ - нагрев PT100", in2 := "Уставки"."Авар Темп контур ГВ")
      Coil( "Авария ГВ контур паст" )
   END_RUNG
   // the same network as SCL:
   "Авария ГВ контур паст" := "fb_AI_Темп ГВ - нагрев PT100" >= "Уставки"."Авар Темп контур ГВ";
END_REGION

REGION Network 9: Звуковой сигнал
   // Управление пищалкой
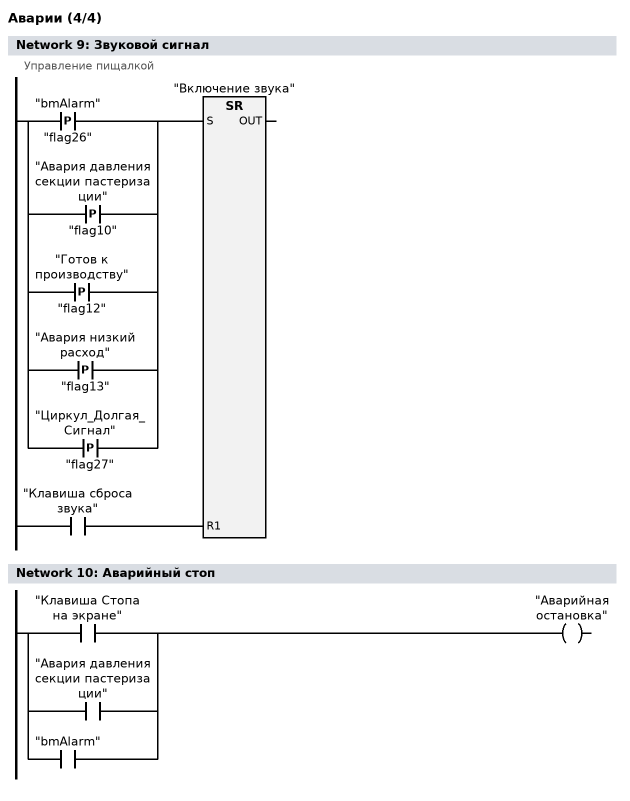
   RUNG wire#powerrail
      P_Contact(operand := "bmAlarm", bit := "flag26")
      wire#w1
      S_SR(operand := "Включение звука", r1 := wire#w2)
   END_RUNG
   RUNG wire#powerrail
      P_Contact(operand := "Авария давления секции пастеризации", bit := "flag10")
   END_RUNG wire#w1
   RUNG wire#powerrail
      P_Contact(operand := "Готов к производству", bit := "flag12")
   END_RUNG wire#w1
   RUNG wire#powerrail
      P_Contact(operand := "Авария низкий расход", bit := "flag13")
   END_RUNG wire#w1
   RUNG wire#powerrail
      P_Contact(operand := "Циркул_Долгая_Сигнал", bit := "flag27")
   END_RUNG wire#w1
   RUNG wire#powerrail
      Contact( "Клавиша сброса звука" )
   END_RUNG wire#w2
   // the same network as SCL:
   #_w1 := "bmAlarm" AND NOT "flag26";   // rising edge of "bmAlarm"
   "flag26" := "bmAlarm";
   #_w2 := "Авария давления секции пастеризации" AND NOT "flag10";   // rising edge of "Авария давления секции пастеризации"
   "flag10" := "Авария давления секции пастеризации";
   #_w3 := "Готов к производству" AND NOT "flag12";   // rising edge of "Готов к производству"
   "flag12" := "Готов к производству";
   #_w4 := "Авария низкий расход" AND NOT "flag13";   // rising edge of "Авария низкий расход"
   "flag13" := "Авария низкий расход";
   #_w5 := "Циркул_Долгая_Сигнал" AND NOT "flag27";   // rising edge of "Циркул_Долгая_Сигнал"
   "flag27" := "Циркул_Долгая_Сигнал";
   IF #_w1 OR #_w2 OR #_w3 OR #_w4 OR #_w5 THEN
       "Включение звука" := TRUE;   // SR flip-flop
   END_IF;
   IF "Клавиша сброса звука" THEN "Включение звука" := FALSE; END_IF;
END_REGION

REGION Network 10: Аварийный стоп
   RUNG wire#powerrail
      Contact( "Клавиша Стопа на экране" )
      wire#w1
      Coil( "Аварийная остановка" )
   END_RUNG
   RUNG wire#powerrail
      Contact( "Авария давления секции пастеризации" )
   END_RUNG wire#w1
   RUNG wire#powerrail
      Contact( "bmAlarm" )
   END_RUNG wire#w1
   // the same network as SCL:
   "Аварийная остановка" := "Клавиша Стопа на экране" OR "Авария давления секции пастеризации" OR "bmAlarm";
END_REGION
END_ORGANIZATION_BLOCK

ORGANIZATION_BLOCK "Wash"   // OB132, LAD, ProgramCycle
TITLE = "Main Program Sweep (Cycle)"
{ S7_Optimized_Access := 'TRUE' }
VERSION : 0.1
   VAR_INPUT
      Initial_Call : Bool;   // Initial call of this OB
      Remanence : Bool;   // =True, if remanent data are available
   END_VAR
   VAR_TEMP
      TimeWash : DInt;
   END_VAR
BEGIN

REGION Network 1
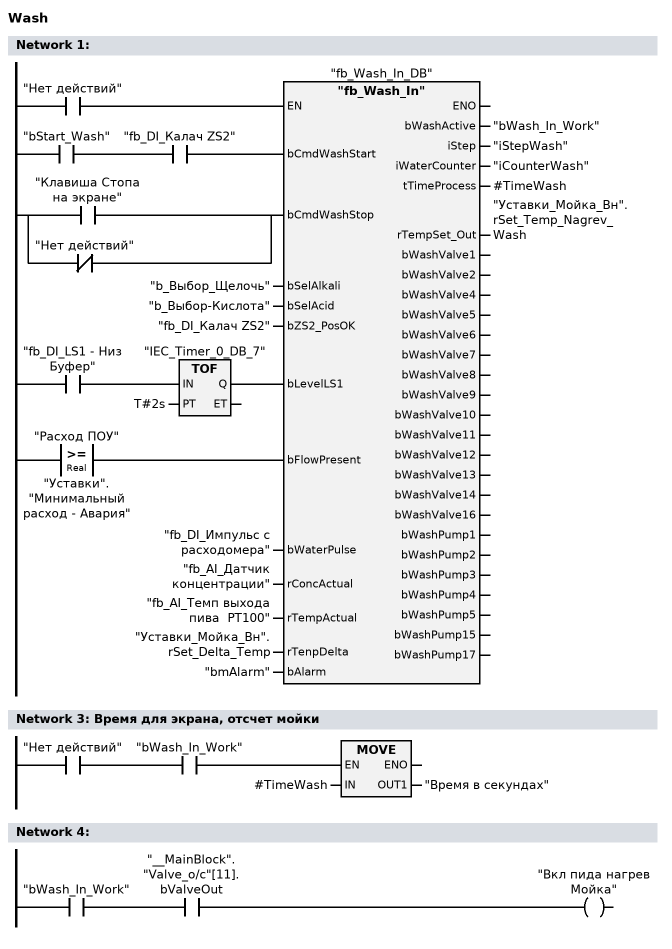
   "IEC_Timer_0_DB_7".TOF(IN := "fb_DI_LS1 - Низ Буфер", PT := T#2s);
   IF "Нет действий" THEN
       "fb_Wash_In_DB"(bCmdWashStart := "bStart_Wash" AND "fb_DI_Калач ZS2",   // "fb_Wash_In"
                       bCmdWashStop := "Клавиша Стопа на экране" OR NOT "Нет действий",
                       bSelAlkali := "b_Выбор_Щелочь",
                       bSelAcid := "b_Выбор-Кислота",
                       bZS2_PosOK := "fb_DI_Калач ZS2",
                       bLevelLS1 := "IEC_Timer_0_DB_7".Q,
                       bFlowPresent := "Расход ПОУ" >= "Уставки"."Минимальный расход - Авария",
                       bWaterPulse := "fb_DI_Импульс с расходомера",
                       rConcActual := "fb_AI_Датчик концентрации",
                       rTempActual := "fb_AI_Темп выхода пива  PT100",
                       rTenpDelta := "Уставки_Мойка_Вн".rSet_Delta_Temp,
                       bAlarm := "bmAlarm",
                       bWashActive => "bWash_In_Work",
                       iStep => "iStepWash",
                       iWaterCounter => "iCounterWash",
                       tTimeProcess => #TimeWash,
                       rTempSet_Out => "Уставки_Мойка_Вн".rSet_Temp_Nagrev_Wash);
   END_IF;
END_REGION

REGION Network 2 (SCL): Время для экрана, отсчет мойки
   "iTime_Min_Wash" := #TimeWash / 60000;
   "iTime_Sec_Wash" :=  #TimeWash / 1000 - "iTime_Min_Wash"*60;
END_REGION

REGION Network 3: Время для экрана, отсчет мойки
   RUNG wire#powerrail
      Contact( "Нет действий" )
      Contact( "bWash_In_Work" )
      Move(in := #TimeWash, out1 => "Время в секундах")
   END_RUNG
   // the same network as SCL:
   IF "Нет действий" AND "bWash_In_Work" THEN "Время в секундах" := #TimeWash; END_IF;
END_REGION

REGION Network 4
   RUNG wire#powerrail
      Contact( "bWash_In_Work" )
      Contact( "__MainBlock"."Valve_o/c"[11].bValveOut )
      Coil( "Вкл пида нагрев Мойка" )
   END_RUNG
   // the same network as SCL:
   "Вкл пида нагрев Мойка" := "bWash_In_Work" AND "__MainBlock"."Valve_o/c"[11].bValveOut;
END_REGION
END_ORGANIZATION_BLOCK

ORGANIZATION_BLOCK "Блоки обработки"   // OB133, LAD, ProgramCycle
TITLE = "Main Program Sweep (Cycle)"
{ S7_Optimized_Access := 'TRUE' }
VERSION : 0.1
   VAR_INPUT
      Initial_Call : Bool;   // Initial call of this OB
      Remanence : Bool;   // =True, if remanent data are available
   END_VAR
BEGIN

REGION Network 1: DI
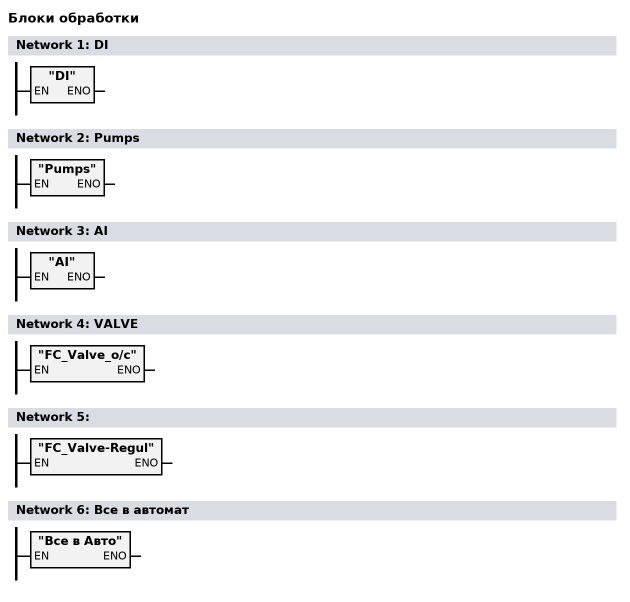
   RUNG wire#powerrail
      "DI"()
   END_RUNG
   // the same network as SCL:
   "DI"();
END_REGION

REGION Network 2: Pumps
   RUNG wire#powerrail
      "Pumps"()
   END_RUNG
   // the same network as SCL:
   "Pumps"();
END_REGION

REGION Network 3: AI
   RUNG wire#powerrail
      "AI"()
   END_RUNG
   // the same network as SCL:
   "AI"();
END_REGION

REGION Network 4: VALVE
   RUNG wire#powerrail
      "FC_Valve_o/c"()
   END_RUNG
   // the same network as SCL:
   "FC_Valve_o/c"();
END_REGION

REGION Network 5
   RUNG wire#powerrail
      "FC_Valve-Regul"()
   END_RUNG
   // the same network as SCL:
   "FC_Valve-Regul"();
END_REGION

REGION Network 6: Все в автомат
   RUNG wire#powerrail
      "Все в Авто"()
   END_RUNG
   // the same network as SCL:
   "Все в Авто"();
END_REGION
END_ORGANIZATION_BLOCK

// folder: AI

FUNCTION_BLOCK "AI_Univ"   // FB3, SCL
{ S7_Optimized_Access := 'TRUE' }
VERSION : 0.1
   VAR_INPUT
      iInValue : Int;   // Значение с модуля сырые
      iTypeSensor : Int;   // 0 - 4-20 $ 1 - RTD Тип датчика
      bSimEnable : Bool;   // Вкл СИМУЛЯЦИЯ
      rSimValue : Real;   // Значение симул
      rHL : Real;   // Нижний предел датчика
      rLL : Real;   // Верхний предел датчика
      bFilterEnable : Bool;   // Включение фильтрации
   END_VAR
   VAR_OUTPUT
      rOut_Value : Real;   // Выходное значение
      bOut_Error : Bool;   // Выход ошибки
   END_VAR
   VAR
      rScaledValue : Real;   // Скалирование датчика
      rFilteredValue : Real;   // Фильтрованное значение датчика
      bRangeError : Bool;   // Выход за пределы - фикс ошибки
      fbFilter : TON_TIME;   // Таймер для фильтра
      tFilter : Time := T#500MS;   // Значение фильтрации
   END_VAR
   VAR CONSTANT
      "Type 4-20" : Int;
      "Type RTD" : Int := 1;
   END_VAR
BEGIN

   // --- Масштабирование ---
   CASE #iTypeSensor OF

       #"Type 4-20":
           #bRangeError := (#iInValue > 30000);

           #rScaledValue := #rLL +(INT_TO_REAL(#iInValue) * (#rHL - #rLL) / 27648.0);

       #"Type RTD":
           // Диагностика обрыва / КЗ / выхода за диапазон
           IF (#iInValue > 32000) OR (#iInValue < -32000) THEN
               #bRangeError := TRUE;
               #rScaledValue := REAL#0.0;
           ELSE
               #rScaledValue := #iInValue / REAL#10.0;   // 0.1 °C
               #bRangeError := FALSE;
           END_IF;

   END_CASE;

   // --- Симуляция ---
   IF #bSimEnable THEN
       #rScaledValue := #rSimValue;
       #bRangeError := FALSE;
   END_IF;

   // --- Фильтрация ---
   IF NOT #bFilterEnable THEN
       #rFilteredValue := #rScaledValue;
   ELSE
       #fbFilter(IN := TRUE,
                 PT := #tFilter);
       IF #fbFilter.Q THEN
           #rFilteredValue := #rScaledValue;
           #fbFilter(IN := FALSE,
                     PT := t#0s);
       END_IF;
   END_IF;

   // --- Выходы ---
   #rOut_Value := #rFilteredValue;
   #bOut_Error := #bRangeError;
END_FUNCTION_BLOCK

FUNCTION_BLOCK "AI_(4-20)_1"   // FB13, LAD
{ S7_Optimized_Access := 'FALSE' }
VERSION : 0.1
   VAR_INPUT
      Input_PLC : Int;   // Вход_Значение на ПЛК
      "HMI_Simulate_on/off" : Bool;   // 0 - выкл, 1 - вкл
      HMI_rSimulate_value : Real;   // значение
      HMI_rParam_Sensor_HL : Real := 16.0;   // Параметры датчика по паспорту (макс значение)bar, C, итд
      HMI_rParam_Sensor_LL : Real;   // Параметры датчика по паспорту (мин значение)bar, C, итд
      "HMI_Filtr_On/off" : Bool;   // Фильтрация, true - вкл
   END_VAR
   VAR_OUTPUT
      Error_out : Bool;   // Ошибка датчика
      HMI_Value_OUT : Real;   // Значение в ед. измерения
   END_VAR
   VAR
      OUT_Scale : Real;   // Выход скалированного значения
      OUT_Normal_Ed : Real;   // Выход нормализованной единицы от 0 др 1
      AI_filtr : "AI_Filtr";
      HMI_Range : Int := 10;   // Кол-во данных для фильтрации
      HMI_iSet_Tik : Int := 2;   // Скорость набора данных для фильтрации
   END_VAR
   VAR_TEMP
      Input_PLC_to_dint : DInt;   // Конвертация из инт в реал
      Error : Word;   // Ошибка в скалировании
      "PLC to_real" : Real;
      value_scale : Real;
      Input_PLC_temp : Int;
      OFF_Param : Bool;
   END_VAR
BEGIN

REGION Network 1
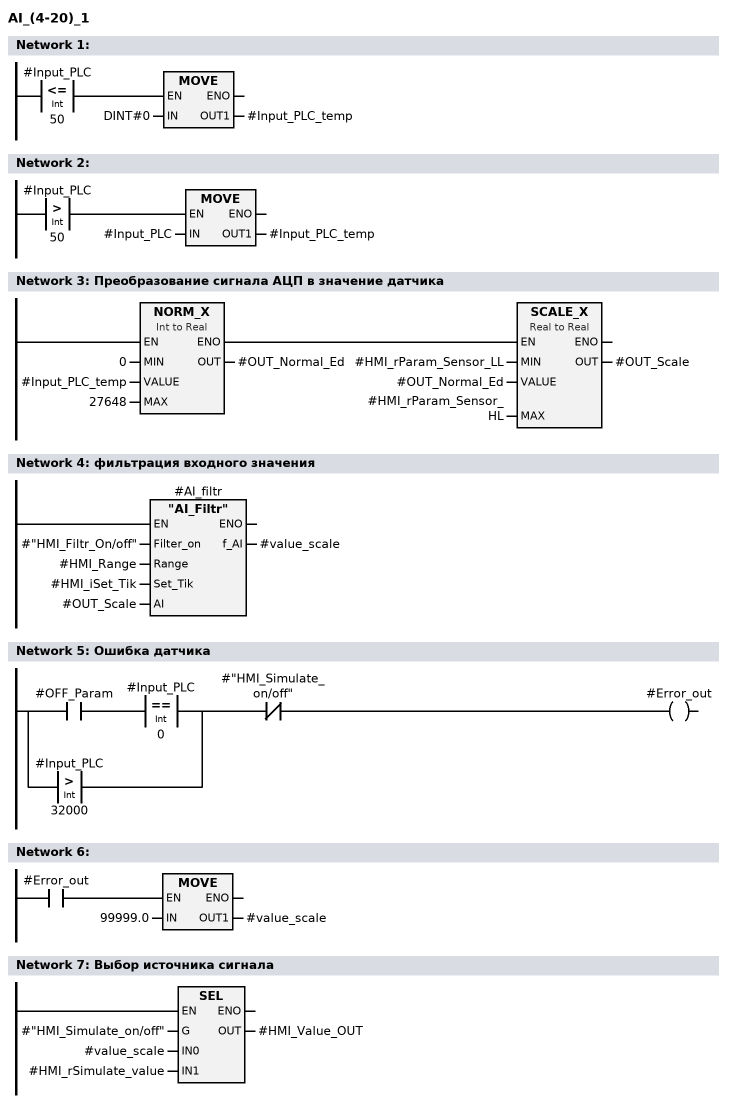
   RUNG wire#powerrail
      { S7_Templates := "SrcType := Int" } LE_Contact(in1 := #Input_PLC, in2 := 50)
      { S7_GenerateENO := "TRUE" } Move(in := DINT#0, out1 => #Input_PLC_temp)
   END_RUNG
   // the same network as SCL:
   IF #Input_PLC <= 50 THEN #Input_PLC_temp := DINT#0; END_IF;
END_REGION

REGION Network 2
   RUNG wire#powerrail
      { S7_Templates := "SrcType := Int" } GT_Contact(in1 := #Input_PLC, in2 := 50)
      { S7_GenerateENO := "TRUE" } Move(in := #Input_PLC, out1 => #Input_PLC_temp)
   END_RUNG
   // the same network as SCL:
   IF #Input_PLC > 50 THEN #Input_PLC_temp := #Input_PLC; END_IF;
END_REGION

REGION Network 3: Преобразование сигнала АЦП в значение датчика
   RUNG wire#powerrail
      { S7_Templates := "[SrcType := Int, DestType := Real]" } Normalize(min := 0, value := #Input_PLC_temp, max := 27648, out => #OUT_Normal_Ed)
      { S7_Templates := "[SrcType := Real, DestType := Real]" } Scale(min := #HMI_rParam_Sensor_LL, value := #OUT_Normal_Ed, max := #HMI_rParam_Sensor_HL, out => #OUT_Scale)
   END_RUNG
   // the same network as SCL:
   #OUT_Normal_Ed := NORM_X(MIN := 0, VALUE := #Input_PLC_temp, MAX := 27648);
   #OUT_Scale := SCALE_X(MIN := #HMI_rParam_Sensor_LL, VALUE := #OUT_Normal_Ed, MAX := #HMI_rParam_Sensor_HL);
END_REGION

REGION Network 4: фильтрация входного значения
   RUNG wire#powerrail
      #AI_filtr(Filter_on := #"HMI_Filtr_On/off", Range := #HMI_Range, Set_Tik := #HMI_iSet_Tik, AI := #OUT_Scale, f_AI => #value_scale)
   END_RUNG
   // the same network as SCL:
   #AI_filtr(Filter_on := #"HMI_Filtr_On/off",   // "AI_Filtr"
             Range := #HMI_Range,
             Set_Tik := #HMI_iSet_Tik,
             AI := #OUT_Scale,
             f_AI => #value_scale);
END_REGION

REGION Network 5: Ошибка датчика
   RUNG wire#powerrail
      Contact( #OFF_Param )
      { S7_Templates := "SrcType := Int" } EQ_Contact(in1 := #Input_PLC, in2 := 0)
      wire#w1
      I_Contact( #"HMI_Simulate_on/off" )
      Coil( #Error_out )
   END_RUNG
   RUNG wire#powerrail
      { S7_Templates := "SrcType := Int" } GT_Contact(in1 := #Input_PLC, in2 := 32000)
   END_RUNG wire#w1
   // the same network as SCL:
   #Error_out := ((#OFF_Param AND (#Input_PLC = 0)) OR (#Input_PLC > 32000)) AND NOT #"HMI_Simulate_on/off";
END_REGION

REGION Network 6
   RUNG wire#powerrail
      Contact( #Error_out )
      Move(in := 99999.0, out1 => #value_scale)
   END_RUNG
   // the same network as SCL:
   IF #Error_out THEN #value_scale := 99999.0; END_IF;
END_REGION

REGION Network 7: Выбор источника сигнала
   #HMI_Value_OUT := SEL(G := #"HMI_Simulate_on/off", IN0 := #value_scale, IN1 := #HMI_rSimulate_value);
END_REGION
END_FUNCTION_BLOCK

FUNCTION_BLOCK "AI_(PT100)"   // FB21, LAD
{ S7_Optimized_Access := 'FALSE' }
VERSION : 0.1
   VAR_INPUT
      Input_PLC : Int;   // Вход_Значение на ПЛК
      "Simulate_on/off" : Bool;   // 0 - выкл, 1 - вкл
      Simulate_value : Real;   // значение
      Param_Sensor_HL : Real := 16.0;   // Параметры датчика по паспорту (макс значение)bar, C, итд
      Param_Sensor_LL : Real;   // Параметры датчика по паспорту (мин значение)bar, C, итд
      "Filtr_On/off" : Bool;   // Фильтрация, true - вкл
   END_VAR
   VAR_OUTPUT
      Value_OUT : Real;   // Значение в ед. измерения
      Error_out : Bool;   // Ошибка датчика
   END_VAR
   VAR
      bipolar : Bool;
      OUT_Scale : Real;   // Выход скалированного значения
      AI_filtr : "AI_Filtr";
      Range : Int := 10;   // Кол-во данных для фильтрации
   END_VAR
   VAR_TEMP
      Input_PLC_to_dint : DInt;   // Конвертация из инт в реал
      Error : Word;   // Ошибка в скалировании
      "PLC to_real" : Real;
      value_scale : Real;
      Input_PLC_temp : Int;
      Input_PLC_to_real : Real;
   END_VAR
BEGIN

REGION Network 1
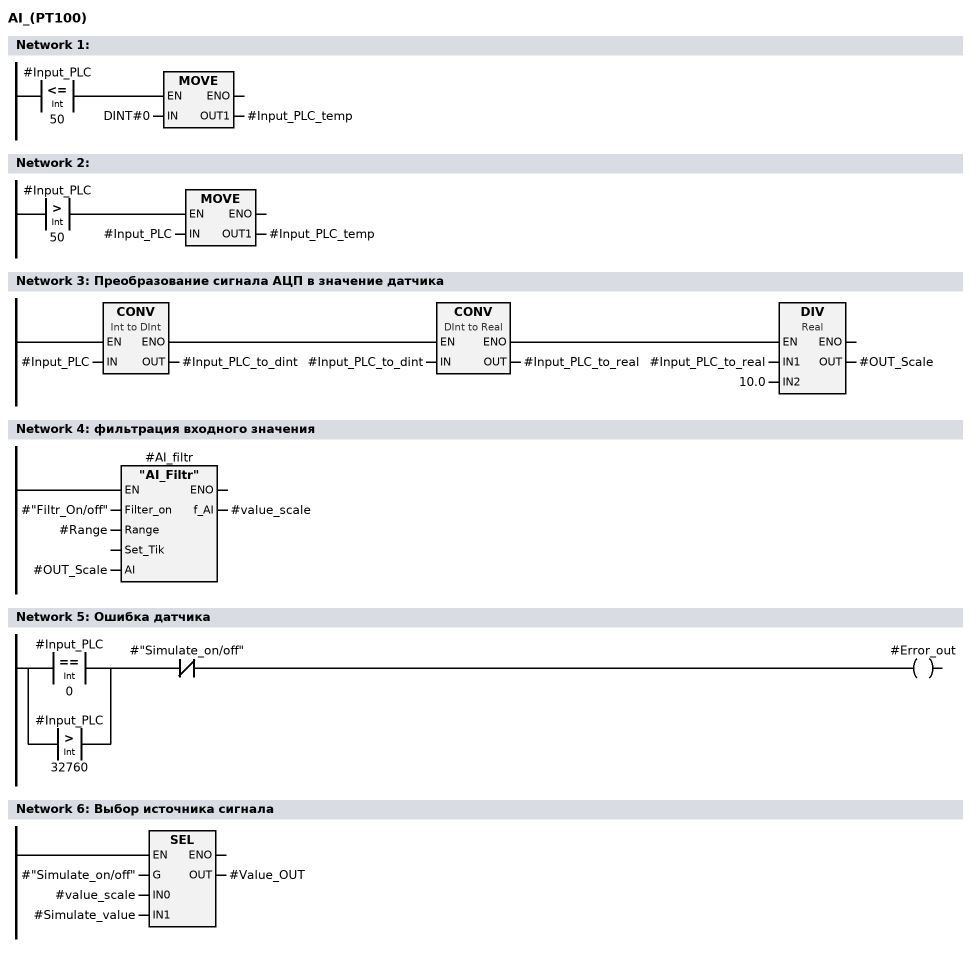
   RUNG wire#powerrail
      { S7_Templates := "SrcType := Int" } LE_Contact(in1 := #Input_PLC, in2 := 50)
      { S7_GenerateENO := "TRUE" } Move(in := DINT#0, out1 => #Input_PLC_temp)
   END_RUNG
   // the same network as SCL:
   IF #Input_PLC <= 50 THEN #Input_PLC_temp := DINT#0; END_IF;
END_REGION

REGION Network 2
   RUNG wire#powerrail
      { S7_Templates := "SrcType := Int" } GT_Contact(in1 := #Input_PLC, in2 := 50)
      { S7_GenerateENO := "TRUE" } Move(in := #Input_PLC, out1 => #Input_PLC_temp)
   END_RUNG
   // the same network as SCL:
   IF #Input_PLC > 50 THEN #Input_PLC_temp := #Input_PLC; END_IF;
END_REGION

REGION Network 3: Преобразование сигнала АЦП в значение датчика
   RUNG wire#powerrail
      { S7_Templates := "[SrcType := Int, DestType := DInt]"; S7_GenerateENO := "TRUE" } Convert(in := #Input_PLC, out => #Input_PLC_to_dint)
      { S7_Templates := "[SrcType := DInt, DestType := Real]"; S7_GenerateENO := "TRUE" } Convert(in := #Input_PLC_to_dint, out => #Input_PLC_to_real)
      { S7_Templates := "SrcType := Real"; S7_GenerateENO := "TRUE" } Div(in1 := #Input_PLC_to_real, in2 := 10.0, out => #OUT_Scale)
   END_RUNG
   // the same network as SCL:
   // ENO of a box is taken as its EN; it also drops when the box reports an error
   #Input_PLC_to_dint := INT_TO_DINT(#Input_PLC);
   #Input_PLC_to_real := DINT_TO_REAL(#Input_PLC_to_dint);
   #OUT_Scale := #Input_PLC_to_real / 10.0;
END_REGION

REGION Network 4: фильтрация входного значения
   RUNG wire#powerrail
      #AI_filtr(Filter_on := #"Filtr_On/off", Range := #Range, Set_Tik :=, AI := #OUT_Scale, f_AI => #value_scale)
   END_RUNG
   // the same network as SCL:
   #AI_filtr(Filter_on := #"Filtr_On/off", Range := #Range, AI := #OUT_Scale, f_AI => #value_scale);   // "AI_Filtr"
END_REGION

REGION Network 5: Ошибка датчика
   RUNG wire#powerrail
      { S7_Templates := "SrcType := Int" } EQ_Contact(in1 := #Input_PLC, in2 := 0)
      wire#w1
      I_Contact( #"Simulate_on/off" )
      Coil( #Error_out )
   END_RUNG
   RUNG wire#powerrail
      { S7_Templates := "SrcType := Int" } GT_Contact(in1 := #Input_PLC, in2 := 32760)
   END_RUNG wire#w1
   // the same network as SCL:
   #Error_out := ((#Input_PLC = 0) OR (#Input_PLC > 32760)) AND NOT #"Simulate_on/off";
END_REGION

REGION Network 6: Выбор источника сигнала
   #Value_OUT := SEL(G := #"Simulate_on/off", IN0 := #value_scale, IN1 := #Simulate_value);
END_REGION
END_FUNCTION_BLOCK

// folder: AI/Funktion

FUNCTION_BLOCK "AI_Filtr"   // FB14, SCL
{ S7_Optimized_Access := 'FALSE' }
VERSION : 0.1
   VAR_INPUT
      Filter_on : Bool;   // Вкл фильтрации
      Range : Int := 10;   // Кол-во входных значений для вычисления среднего
      Set_Tik : Int := 2;   // Задача периода фильтрации от 1(мин) до 8
      AI : Real;   // Вход значения датчика
   END_VAR
   VAR_OUTPUT
      f_AI : Real;   // выход значения с фильтром или без
   END_VAR
   VAR
      CTU : CTU_INT;   // счетчик для подсчета кол-во вх значений
      Tik : Bool;   // Время фильтрации
      ai_array : Array[0..#Max_Array] of Real;   // Массив значений датчика
      i : Int;   // для цикла ФОР
      sum_AI : Real;   // Суммирование значений с входа датчика
      Avarage_AI : Real;   // Среднее значение датчика
      fRS_set : Bool;   // Для RS тригера
      fRS_res : Bool;   // Для RS тригера
      fRS_out : Bool;   // Для RS тригера
      FullFiltr : Bool;   // Ожидание наполнения значений для вычисления средней
      Res_count : Bool;   // сброс счетчика
   END_VAR
   VAR CONSTANT
      Max_Array : Int := 30;   // Размер массива
   END_VAR
BEGIN

   CASE #Set_Tik OF                   
       1:  
           #Tik := "Time_0.1s";
       2:  
           #Tik := "Time_0.2s";
       3:
           #Tik := "Time_0.4s";
       4:
           #Tik := "Time_0.5s";
       5:
           #Tik := "Time_0.8s";
       6:
           #Tik := "Time_1s";
       7:
           #Tik := "Time_1.6s";
       8:
           #Tik := "Time_2s";
       0:
           #Tik := "Time_0.1s";

       ELSE  
           #Set_Tik := 8;
   END_CASE;  // Выбор периода фильтрации входного сигнала
   REGION RS триггер
       IF #fRS_set THEN
           #fRS_out := true;
       ELSIF #fRS_res AND NOT #fRS_set THEN
           #fRS_out := false;
       END_IF;
   END_REGION

   REGION Подсчет среднего значения входа
       // Statement section REGION
           #CTU(CU := #Tik,
                PV := #Range,
                R := #Res_count,
                Q => #Res_count);                                      // Счетчик для набора значений с входа
           #ai_array[#CTU.CV] := #AI;                                  // Запись значений с входа в массив

           IF #Res_count THEN                                              // СБРОС как счетчик переполниться Для корректной работы счетчика
               #i := 0;
               #sum_AI := 0;
           END_IF;

           IF #Range <> #i THEN                                    // выход из цикла FOR при суммировании всех значений, почему то сам не прекращел подсчет при окончании цикла все время суммировался 
               FOR #i := 0 TO (#Range - 1) DO
                   #sum_AI := #ai_array[#i] + #sum_AI;             // суммирование значений
               END_FOR;
           END_IF;

       #Avarage_AI := #sum_AI / #Range;                             // Вычисление среднего значения
       #fRS_res := NOT #Filter_on;

   END_REGION

   REGION Выбор выхода прямое или фильтрованное значение
       IF #Filter_on THEN                                          //Включение выключение фильтрации
           #fRS_set := #CTU.QD;                                    //При включении фильтра ждем наполнения значениями с входа, пока ждем - отправляем на выход прямое значение входа, далее фильтруем
            #FullFiltr := #fRS_out;

          IF #FullFiltr THEN                                       //Когда фильтр наполнился - вывыодим среднее значение входа
               #f_AI := #Avarage_AI;                              // ЗАпись значения на выход AI
          ELSE
               #f_AI := #AI;                                     // Прямой вывод значения, пока значения не наполнились данными
          END_IF;
       ELSE
           #f_AI := #AI;                                        // Если фильтр выключен, на выход прямое значение с входа
       END_IF; 

   END_REGION
END_FUNCTION_BLOCK

FUNCTION "Calculate_AI" : Void   // FC7, SCL
{ S7_Optimized_Access := 'FALSE' }
VERSION : 0.1
   VAR_INPUT
      IN_sensors : Int;
      Current_max : Real;
      Current_min : Real;
      Code_HL : Real;
      Code_LL : Real;
      Param_Sensor_HL : Real;   // Параметры датчика по паспорту (макс значение)bar, C, итд
      Param_Sensor_LL : Real;   // Параметры датчика по паспорту (мин значение)bar, C, итд
   END_VAR
   VAR_OUTPUT
      signal_Electric : Real;   // выход в электрических ед измерения
      Value_Sensor : Real;   // выход реального значения датчика в ед измерения
   END_VAR
   VAR_TEMP
      sensor_to_real : Real;   // Для конвертации INT to Real
      result_to_out_signal : Real;   // Для вычитания реального значения показания датчика
   END_VAR
BEGIN
       //Convert int to real
   #sensor_to_real := INT_TO_REAL(#IN_sensors);

       // Расчет значения АЦП контроллера в значение эл. ед измерения (I, U) в зависимости от значений на входе
   #signal_Electric := ((#sensor_to_real - #Code_LL) * (#Current_max - #Current_min) / (#Code_HL - #Code_LL))+ #Current_min;
   #result_to_out_signal := #signal_Electric;

   // Расчет значения в реальных единицах измерения датчика (bar, C,) в зависимости от введеных параметров датчика Param_Sensor min/max
   #Value_Sensor := (#result_to_out_signal - #Current_min) * (#Param_Sensor_HL - #Param_Sensor_LL) / (#Current_max - #Current_min) + #Param_Sensor_LL;
END_FUNCTION

// folder: DI

FUNCTION_BLOCK "DI_fb_Arrey_Old"   // FB1, SCL
{ S7_Optimized_Access := 'TRUE' }
VERSION : 0.1
   VAR_IN_OUT
      aDI : Array[*] of "ty_DI";
   END_VAR
   VAR
      aTON_Filtr : Array[0..50] of TON_TIME;   // Следить за кол-вом DI
      bTonIn : Bool;
      Volue : Bool;
   END_VAR
   VAR_TEMP
      i : Int;
      SizeArrey : Int;   // Размер массива
   END_VAR
   VAR CONSTANT
      n : Int := 10;
   END_VAR
BEGIN
   #SizeArrey := UPPER_BOUND(ARR := #aDI, DIM := 1);

   // Цикл перебор значений - кол-во DI входов (строго дожно быть = массиву, не больше, меньш можно, больше ошибка)
   FOR #i := 0 TO #SizeArrey DO

       REGION Таймер фильтрации входа
           // управление таймером 
           #bTonIn := NOT #aDI[#i].Sim AND #aDI[#i].Filtr AND #aDI[#i].In;
           // вызов таймера фильтрации
           #aTON_Filtr[#i](IN := #bTonIn,
                           PT := #aDI[#i].TimeFiltr);
       END_REGION



       //-------------Условие симуляции, если да работает только по сигналам симулирования 
       IF (#aDI[#i].Sim = TRUE) THEN
           #Volue := #aDI[#i].Sim_Out;

       //------------Условие если фильтрация включена--------------------
       ELSIF #aDI[#i].Filtr = TRUE THEN

           #Volue := #aTON_Filtr[#i].Q;    //Выход по таймеру значения таймера

       ELSE
           #Volue := #aDI[#i].In;

       END_IF;

       //Присвоение выходу значения
       #aDI[#i].Out :=  #Volue;



   END_FOR;
END_FUNCTION_BLOCK

FUNCTION_BLOCK "DI_fb_Arrey"   // FB11, SCL
{ S7_Optimized_Access := 'TRUE' }
VERSION : 0.1
   VAR_IN_OUT
      aDI : Array[*] of "ty_DI";
   END_VAR
   VAR
      aTON_Filtr : Array[0..50] of TON_TIME;   // Следить за кол-вом DI
      bTonIn : Bool;
      Volue : Bool;
   END_VAR
   VAR_TEMP
      i : Int;
      SizeArrey : Int;   // Размер массива
   END_VAR
   VAR CONSTANT
      n : Int := 10;
   END_VAR
BEGIN
   #SizeArrey := UPPER_BOUND(ARR := #aDI, DIM := 1);

   // Цикл перебор значений - кол-во DI входов (строго дожно быть = массиву, не больше, меньш можно, больше ошибка)
   IF #i >= 5 THEN
   #i := 0;
   END_IF;

       REGION Таймер фильтрации входа
           // управление таймером 
           #bTonIn := NOT #aDI[#i].Sim AND #aDI[#i].Filtr AND #aDI[#i].In;
           // вызов таймера фильтрации
           #aTON_Filtr[#i](IN := #bTonIn,
                           PT := #aDI[#i].TimeFiltr);
       END_REGION



       //-------------Условие симуляции, если да работает только по сигналам симулирования 
       IF (#aDI[#i].Sim = TRUE) THEN
           #Volue := #aDI[#i].Sim_Out;

       //------------Условие если фильтрация включена--------------------
       ELSIF #aDI[#i].Filtr = TRUE THEN

           #Volue := #aTON_Filtr[#i].Q;    //Выход по таймеру значения таймера

       ELSE
           #Volue := #aDI[#i].In;

       END_IF;

       //Присвоение выходу значения
       #aDI[#i].Out :=  #Volue;

       #i := #i + 1;
END_FUNCTION_BLOCK

// folder: Pumps

FUNCTION_BLOCK "FB_Pump"   // FB2, SCL
{ S7_Optimized_Access := 'FALSE' }
VERSION : 0.1
   VAR_INPUT
      bManualMode : Bool;   // Выбор ручного режима
      bManualStart : Bool;   // Ручной режим - старт
      bManualStop : Bool;   // Ручной режим - стоп
      rManualSpeed : Real;   // Ручной режим - скорость
      bDryRunn : Bool;   // Защита от сухого хода
      bAutoSTop : Bool;   // Остановка насоса
      bAutoStartPerm : Bool;   // Команда на работоу в авто режиме
      rAutoSpeed : Real;   // Скорость в авто режиме
      bАвтоматы : Bool;   // Готовность привода (автоматы)
      bПускатели : Bool;   // Готовность Пускателя
      bDriveRunning : Bool;   // Привод в работе
      bDriveFault : Bool;   // Привод в ошибке
      rMinSpeed : Real;   // Минимальная скорость
      rMaxSpeed : Real := 100.0;   // Максимальная скорость
      bResetFault : Bool;   // Сброс аварии
   END_VAR
   VAR_OUTPUT
      bRunCmd : Bool;   // Пуск частотника
      iSpeedOut : Int;   // Скорость насоса для аналогового выхода
      "rSpeedHMI(0-100)" : Real;   // Скорость работы (0-100) для HMI
      bPumpRunning : Bool;   // Работа
      bPumpFault : Bool;   // Авария
      iStatus : Int;   // Статус (0 - стоп 1 - работа 2 - авария)
   END_VAR
   VAR
      bFaultLatch : Bool;
      bRunRequest : Bool;
      rSpeedPump : Real;   // Скорость насоса
      TON_NotStartRun : TON_TIME;   // ТАймер ожидания сигнала о запуске
      TON_NotContactRun : TON_TIME;   // ТАймер ожидания с контактора
      TON_DryRun : TON_TIME;   // Таймер сухого хода
   END_VAR
BEGIN
   (*
   // 1. Обработка аварий
   // Обработка ожидания сигнала о работе после старта
   IF #bAutoStartPerm THEN
       ;

   END_IF;
   *)

   // 1 Ручной режим
   IF #bManualMode THEN
       // Ручной режим
       IF #bManualStart THEN
           #bRunRequest := TRUE;
       ELSE
           #bRunRequest := FALSE;
       END_IF;
   ELSE
       // Автоматический режим
       // 
       //Обработка аварий
       //--------------------------------------------------------------------------------------------------------
       IF #bAutoStartPerm THEN
           #TON_NotStartRun(IN := NOT #bDriveRunning,PT := t#5s);  //Таймер ожидания сигнала подтверждения пуска от частотника
           #TON_NotContactRun(IN := NOT #bПускатели, PT := t#10s);  //Таймер ожидания сигнала подтверждения пуска от пускателя
           #TON_DryRun(IN:= NOT #bDryRunn, PT := t#10s);    //Таймер ожидания останова по сухому ходу

       ELSE
           #TON_NotStartRun(IN :=FALSE,PT := t#5s);
           #TON_NotContactRun(IN := FALSE,PT := t#5s);
       END_IF;
       #bFaultLatch := #TON_NotStartRun.Q OR #TON_NotContactRun.Q OR (#bDriveFault OR NOT #bАвтоматы) OR (NOT #bResetFault AND #bFaultLatch); //Разкоментировать если нужна будет фиксация АЛАРМА, сброс только по входу РЕСЕТ
       #bPumpFault := #bFaultLatch;

       //Старт--------------------------------
       #bRunRequest := #bAutoStartPerm AND NOT #bPumpFault AND NOT #TON_DryRun.Q;
   END_IF;

   // 3. Задание скорости
   IF #bManualMode THEN
       #"rSpeedHMI(0-100)" := LIMIT(MN := #rMinSpeed, IN := #rManualSpeed, MX := #rMaxSpeed);
   ELSE
       #"rSpeedHMI(0-100)" := LIMIT(MN := #rMinSpeed, IN := #rAutoSpeed, MX := #rMaxSpeed);
   END_IF;

   // Преобразование значения от 0-100 до 0-27648 для аналогового выхода
   #iSpeedOut := REAL_TO_INT((#"rSpeedHMI(0-100)"/ 100.0) * 27648.0);

   // 4. Выходные команды и статусы
   // Команды старт
   #bRunCmd := #bRunRequest;

   //Выход статуса для HMI
   #bPumpRunning := #bDriveRunning AND #bRunCmd OR (#bManualStart AND #bManualMode);



   // 5. Числовой статус (для HMI/SCADA)
   IF #bFaultLatch THEN
       #iStatus := 2; // Авария
   ELSIF #bPumpRunning THEN
       #iStatus := 1; // Работа
   ELSE
       #iStatus := 0; // Стоп
   END_IF;

   IF NOT #bAutoStartPerm AND NOT #bManualMode THEN
       #bRunCmd := FALSE;
   END_IF;
END_FUNCTION_BLOCK

// folder: Valve_o/c

FUNCTION_BLOCK "Valve_o/c_fb_Arrey_old"   // FB4, SCL
{ S7_Optimized_Access := 'TRUE' }
VERSION : 0.1
   VAR_IN_OUT
      aValve : Array[*] of "ty_Valve";
   END_VAR
   VAR
      aOpenTimer : Array[0..#Size_Timer] of TON_TIME;   // Кол-во таймеров должно быть больше кол-ва клапанов - смотри в КОНСТАНТАХ
      aEnableTimer : Array[0..#Size_Timer] of Bool;   // Кол-во таймеров должно быть больше кол-ва клапанов - смотри в КОНСТАНТАХ
      aWaitingOpen : Array[0..#Size_Timer] of Bool;   // Кол-во таймеров должно быть больше кол-ва клапанов - смотри в КОНСТАНТАХ
      i : Int;
      SizeArray : Int;
   END_VAR
   VAR CONSTANT
      Size_Timer : Int := 50;   // Обязательно котнтроллировать размер массива должно быть больше кол-ва клапанов
   END_VAR
BEGIN

   // .........-------ОБЯЗАТЕЛЬНО КОНТРОЛЛИРОВАТЬ РАЗМЕР МАССИВА ДЛЯ ТАЙМЕРА - ДОЛЖННО БЫТЬ СТРОГО БОЛЬШЕ ВХОДНОГО МАССИВА ИНАЧЕ НЕ БУДЕТ РАБОТАТЬ!!!!!-------............
   // Size_Array - CONSTANTA = СМОТРИ В РАЗДЕЛЕ КОНСТАНТ

   #SizeArray := UPPER_BOUND(ARR := #aValve, DIM := 1);


   FOR #i := 1 TO #SizeArray DO

       // ==================================================
       // ОБНОВЛЕНИЕ ТАЙМЕРА (ВСЕГДА)
       // ==================================================
       #aOpenTimer[#i](
                       IN := #aEnableTimer[#i],
                       PT := #aValve[#i].tMaxTime * 1000
       );

       // ==================================================
       // СБРОС АВАРИИ
       // ==================================================
       IF #aValve[#i].bResetAlarm THEN
           #aValve[#i].bValveFault := FALSE;
           #aWaitingOpen[#i] := FALSE;
           #aEnableTimer[#i] := FALSE;
       END_IF;

       // ==================================================
       // РЕЖИМ РУЧНОЙ
       // ==================================================
       IF #aValve[#i].bManualMode THEN

           #aValve[#i].bValveOut := #aValve[#i].bManualOpen;
           #aValve[#i].bValveFault := FALSE;
           #aEnableTimer[#i] := FALSE;
           #aWaitingOpen[#i] := FALSE;

           // ==================================================
           // РЕЖИМ АВТО
           // ==================================================
       ELSE

           // --- Управление выходом ---
           IF #aValve[#i].bAuto_OpenCmd AND NOT #aValve[#i].bValveFault THEN
               #aValve[#i].bValveOut := TRUE;
           ELSE
               #aValve[#i].bValveOut := FALSE;
           END_IF;

           // --- Контроль обратной связи ---
           IF #aValve[#i].bHaveFeedback THEN

               IF #aValve[#i].bAuto_OpenCmd
                   AND NOT #aValve[#i].bFeedbackOpen
                   AND NOT #aValve[#i].bValveFault THEN

                   #aEnableTimer[#i] := TRUE;
                   #aWaitingOpen[#i] := TRUE;

               ELSE
                   #aEnableTimer[#i] := FALSE;

                   IF #aValve[#i].bFeedbackOpen THEN
                       #aWaitingOpen[#i] := FALSE;
                   END_IF;
               END_IF;

           ELSE
               #aEnableTimer[#i] := FALSE;
           END_IF;

           // --- Авария по таймеру ---
           IF #aOpenTimer[#i].Q AND #aWaitingOpen[#i] THEN
               #aValve[#i].bValveFault := TRUE;
               #aWaitingOpen[#i] := FALSE;
               #aEnableTimer[#i] := FALSE;
           END_IF;

       END_IF;

       // ==================================================
       // СОСТОЯНИЕ КЛАПАНА
       // ==================================================
       IF #aValve[#i].bValveFault THEN
           #aValve[#i].iValveState := 2;   // авария
       ELSIF #aValve[#i].bHaveFeedback AND #aValve[#i].bFeedbackOpen THEN
           #aValve[#i].iValveState := 1;   // открыт
       ELSIF NOT #aValve[#i].bHaveFeedback AND
           ((NOT #aValve[#i].bManualMode AND #aValve[#i].bAuto_OpenCmd)
           OR (#aValve[#i].bManualMode AND #aValve[#i].bManualOpen)) THEN
           #aValve[#i].iValveState := 1;   // открыт
       ELSE
           #aValve[#i].iValveState := 0;   // закрыт
       END_IF;

   END_FOR;
END_FUNCTION_BLOCK

FUNCTION_BLOCK "Valve_o/c_fb_Arrey"   // FB9, SCL
{ S7_Optimized_Access := 'TRUE' }
VERSION : 0.1
   VAR_IN_OUT
      aValve : Array[*] of "ty_Valve";
   END_VAR
   VAR
      aOpenTimer : Array[0..#Size_Timer] of TON_TIME;   // Кол-во таймеров должно быть больше кол-ва клапанов - смотри в КОНСТАНТАХ
      aEnableTimer : Array[0..#Size_Timer] of Bool;   // Кол-во таймеров должно быть больше кол-ва клапанов - смотри в КОНСТАНТАХ
      aWaitingOpen : Array[0..#Size_Timer] of Bool;   // Кол-во таймеров должно быть больше кол-ва клапанов - смотри в КОНСТАНТАХ
      i : Int;
      SizeArray : Int;
   END_VAR
   VAR CONSTANT
      Size_Timer : Int := 50;   // Обязательно котнтроллировать размер массива должно быть больше кол-ва клапанов
   END_VAR
BEGIN

   // .........-------ОБЯЗАТЕЛЬНО КОНТРОЛЛИРОВАТЬ РАЗМЕР МАССИВА ДЛЯ ТАЙМЕРА - ДОЛЖННО БЫТЬ СТРОГО БОЛЬШЕ ВХОДНОГО МАССИВА ИНАЧЕ НЕ БУДЕТ РАБОТАТЬ!!!!!-------............
   // Size_Array - CONSTANTA = СМОТРИ В РАЗДЕЛЕ КОНСТАНТ

   #SizeArray := UPPER_BOUND(ARR := #aValve, DIM := 1);
   IF #i >= #SizeArray THEN
       #i := 1;
   END_IF;


       // ==================================================
       // ОБНОВЛЕНИЕ ТАЙМЕРА (ВСЕГДА)
       // ==================================================
       #aOpenTimer[#i](
                       IN := #aEnableTimer[#i],
                       PT := #aValve[#i].tMaxTime * 1000
       );

       // ==================================================
       // СБРОС АВАРИИ
       // ==================================================
       IF #aValve[#i].bResetAlarm THEN
           #aValve[#i].bValveFault := FALSE;
           #aWaitingOpen[#i] := FALSE;
           #aEnableTimer[#i] := FALSE;
       END_IF;

       // ==================================================
       // РЕЖИМ РУЧНОЙ
       // ==================================================
       IF #aValve[#i].bManualMode THEN

           #aValve[#i].bValveOut := #aValve[#i].bManualOpen;
           #aValve[#i].bValveFault := FALSE;
           #aEnableTimer[#i] := FALSE;
           #aWaitingOpen[#i] := FALSE;

           // ==================================================
           // РЕЖИМ АВТО
           // ==================================================
       ELSE

           // --- Управление выходом ---
           IF #aValve[#i].bAuto_OpenCmd AND NOT #aValve[#i].bValveFault THEN
               #aValve[#i].bValveOut := TRUE;
           ELSE
               #aValve[#i].bValveOut := FALSE;
           END_IF;

           // --- Контроль обратной связи ---
           IF #aValve[#i].bHaveFeedback THEN

               IF #aValve[#i].bAuto_OpenCmd
                   AND NOT #aValve[#i].bFeedbackOpen
                   AND NOT #aValve[#i].bValveFault THEN

                   #aEnableTimer[#i] := TRUE;
                   #aWaitingOpen[#i] := TRUE;

               ELSE
                   #aEnableTimer[#i] := FALSE;

                   IF #aValve[#i].bFeedbackOpen THEN
                       #aWaitingOpen[#i] := FALSE;
                   END_IF;
               END_IF;

           ELSE
               #aEnableTimer[#i] := FALSE;
           END_IF;

           // --- Авария по таймеру ---
           IF #aOpenTimer[#i].Q AND #aWaitingOpen[#i] THEN
               #aValve[#i].bValveFault := TRUE;
               #aWaitingOpen[#i] := FALSE;
               #aEnableTimer[#i] := FALSE;
           END_IF;

       END_IF;

       // ==================================================
       // СОСТОЯНИЕ КЛАПАНА
       // ==================================================
       IF #aValve[#i].bValveFault THEN
           #aValve[#i].iValveState := 2;   // авария
       ELSIF #aValve[#i].bHaveFeedback AND #aValve[#i].bFeedbackOpen THEN
           #aValve[#i].iValveState := 1;   // открыт
       ELSIF NOT #aValve[#i].bHaveFeedback AND
           ((NOT #aValve[#i].bManualMode AND #aValve[#i].bAuto_OpenCmd)
           OR (#aValve[#i].bManualMode AND #aValve[#i].bManualOpen)) THEN
           #aValve[#i].iValveState := 1;   // открыт
       ELSE
           #aValve[#i].iValveState := 0;   // закрыт
       END_IF;

       #i := #i + 1;
END_FUNCTION_BLOCK